SPLINE
SPL {X  -140.007, Y  +297.383, Z    +0.000, E1   +42.766, E3 +239231.187}
SPL {X  -156.919, Y  +337.064, Z    +0.000, E1   +27.647, E3 +239237.338}
SPL {X  -160.736, Y  +354.534, Z    +0.000, E1   +18.553, E3 +239240.033}
SPL {X  -162.078, Y  +364.978, Z    +0.000, E1   +12.369, E3 +239241.718}
SPL {X  -162.752, Y  +375.778, Z    +0.000, E1    +5.236, E3 +239241.427}
SPL {X  -162.820, Y  +381.939, Z    +0.000, E1    +0.593, E3 +239241.054}
SPL {X  -162.820, Y  +383.993, Z    +0.000, E1    -1.497, E3 +239240.627}
SPL {X  -162.820, Y  +388.628, Z    +0.000, E1    -7.678, E3 +239240.530}
SPL {X  -162.820, Y  +394.643, Z    +0.000, E1   -17.317, E3 +239240.330}
SPL {X  -162.820, Y  +401.515, Z    +0.000, E1   -27.960, E3 +239241.150}
SPL {X  -162.820, Y  +415.147, Z    +0.000, E1   -45.856, E3 +239240.466}
SPL {X  -162.820, Y  +437.881, Z    +0.000, E1   -59.335, E3 +239245.884}
SPL {X  -162.820, Y  +475.967, Z    +0.000, E1   -65.140, E3 +239263.337}
SPL {X  -162.820, Y  +578.686, Z    +0.000, E1   -67.085, E3 +239331.578}
ENDSPLINE

SPLINE
SPL {X  -162.820, Y  +565.364, Z    +0.000, E1   -63.589, E3 +239345.578}
ENDSPLINE

SPLINE
SPL {X  -162.820, Y  +574.608, Z    +0.000, E1   -63.370, E3 +239356.837}
SPL {X  -162.820, Y  +584.314, Z    +0.000, E1   -63.342, E3 +239367.129}
SPL {X  -162.820, Y  +593.857, Z    +0.000, E1   -63.382, E3 +239376.831}
SPL {X  -162.820, Y  +602.272, Z    +0.000, E1   -63.279, E3 +239386.359}
SPL {X  -162.820, Y  +613.309, Z    +0.000, E1   -63.489, E3 +239396.358}
SPL {X  -162.820, Y  +619.956, Z    +0.000, E1   -63.110, E3 +239406.044}
SPL {X  -162.820, Y  +634.513, Z    +0.000, E1   -63.471, E3 +239418.810}
SPL {X  -162.820, Y  +648.936, Z    +0.000, E1   -63.278, E3 +239435.265}
SPL {X  -162.820, Y  +662.662, Z    +0.000, E1   -63.383, E3 +239448.757}
SPL {X  -162.819, Y  +673.983, Z    +0.000, E1   -63.398, E3 +239460.480}
SPL {X  -162.399, Y  +685.202, Z    +0.000, E1   -63.235, E3 +239473.474}
SPL {X  -161.289, Y  +695.772, Z    +0.000, E1   -63.167, E3 +239484.924}
SPL {X  -160.212, Y  +702.527, Z    +0.000, E1   -62.898, E3 +239493.905}
SPL {X  -158.647, Y  +710.128, Z    +0.000, E1   -62.776, E3 +239502.727}
SPL {X  -156.957, Y  +716.799, Z    +0.000, E1   -62.460, E3 +239511.845}
SPL {X  -154.447, Y  +725.041, Z    +0.000, E1   -62.170, E3 +239522.503}
SPL {X  -151.721, Y  +732.586, Z    +0.000, E1   -61.616, E3 +239533.752}
SPL {X  -149.420, Y  +738.185, Z    +0.000, E1   -61.282, E3 +239541.642}
SPL {X  -146.033, Y  +745.504, Z    +0.000, E1   -60.844, E3 +239551.909}
SPL {X  -142.518, Y  +752.234, Z    +0.000, E1   -60.144, E3 +239562.535}
SPL {X  -139.430, Y  +757.582, Z    +0.000, E1   -59.554, E3 +239571.067}
SPL {X  -134.550, Y  +765.187, Z    +0.000, E1   -59.954, E3 +239577.018}
SPL {X  -102.851, Y  +799.722, Z    +0.000, E1   -53.923, E3 +239667.511}
SPL {X  -101.618, Y  +800.716, Z    +0.000, E1   -52.212, E3 +239780.496}
ENDSPLINE

SPLINE
SPL {X  -141.567, Y  +753.931, Z    +0.000, E1   -42.659, E3 +239817.198}
SPL {X  -155.442, Y  +721.958, Z    +0.000, E1   -30.769, E3 +239824.104}
SPL {X  -161.417, Y  +694.832, Z    +0.000, E1   -16.464, E3 +239828.073}
SPL {X  -162.580, Y  +682.344, Z    +0.000, E1    -8.212, E3 +239828.280}
SPL {X  -162.811, Y  +675.182, Z    +0.000, E1    -3.078, E3 +239828.313}
SPL {X  -162.820, Y  +671.474, Z    +0.000, E1    -0.022, E3 +239827.783}
SPL {X  -162.820, Y  +668.525, Z    +0.000, E1    +3.543, E3 +239827.476}
SPL {X  -162.820, Y  +663.189, Z    +0.000, E1   +11.952, E3 +239827.465}
SPL {X  -162.820, Y  +655.445, Z    +0.000, E1   +24.952, E3 +239827.412}
SPL {X  -162.820, Y  +644.088, Z    +0.000, E1   +41.840, E3 +239827.548}
SPL {X  -162.820, Y  +632.645, Z    +0.000, E1   +53.114, E3 +239828.283}
SPL {X  -162.820, Y  +584.142, Z    +0.000, E1   +66.966, E3 +239843.626}
SPL {X  -162.820, Y  +471.906, Z    +0.000, E1   +66.781, E3 +239925.868}
SPL {X  -162.820, Y  +470.218, Z    +0.000, E1   +64.979, E3 +239941.868}
SPL {X  -162.820, Y  +452.619, Z    +0.000, E1   +64.912, E3 +239959.546}
SPL {X  -162.820, Y  +437.579, Z    +0.000, E1   +64.893, E3 +239974.228}
SPL {X  -162.820, Y  +425.248, Z    +0.000, E1   +64.950, E3 +239985.816}
SPL {X  -162.820, Y  +417.868, Z    +0.000, E1   +64.478, E3 +239996.634}
ENDSPLINE

SPLINE
SPL {X  -162.820, Y  +442.889, Z    +0.000, E1   +58.918, E3 +240008.814}
ENDSPLINE

SPLINE
SPL {X  -162.820, Y  +428.091, Z    +0.000, E1   +59.583, E3 +240022.587}
SPL {X  -162.820, Y  +410.436, Z    +0.000, E1   +60.611, E3 +240036.788}
SPL {X  -162.820, Y  +385.611, Z    +0.000, E1   +62.089, E3 +240054.686}
ENDSPLINE

SPLINE
SPL {X  -162.820, Y  +397.122, Z    +0.000, E1   +58.099, E3 +240067.658}
ENDSPLINE

SPLINE
SPL {X  -162.820, Y  +387.359, Z    +0.000, E1   +58.365, E3 +240078.519}
SPL {X  -162.810, Y  +378.731, Z    +0.000, E1   +58.366, E3 +240089.577}
SPL {X  -162.546, Y  +371.051, Z    +0.000, E1   +58.239, E3 +240100.297}
SPL {X  -161.863, Y  +362.875, Z    +0.000, E1   +58.273, E3 +240110.522}
SPL {X  -161.159, Y  +357.301, Z    +0.000, E1   +57.946, E3 +240119.822}
SPL {X  -159.864, Y  +349.614, Z    +0.000, E1   +57.922, E3 +240129.898}
SPL {X  -158.300, Y  +342.404, Z    +0.000, E1   +57.579, E3 +240141.344}
SPL {X  -156.187, Y  +334.499, Z    +0.000, E1   +57.331, E3 +240153.004}
SPL {X  -154.237, Y  +328.333, Z    +0.000, E1   +56.930, E3 +240163.214}
SPL {X  -152.732, Y  +324.078, Z    +0.000, E1   +56.482, E3 +240171.219}
SPL {X  -150.609, Y  +318.634, Z    +0.000, E1   +56.366, E3 +240178.913}
SPL {X  -148.206, Y  +313.080, Z    +0.000, E1   +55.888, E3 +240188.625}
SPL {X  -145.956, Y  +308.339, Z    +0.000, E1   +55.380, E3 +240197.301}
SPL {X  -143.330, Y  +303.254, Z    +0.000, E1   +55.057, E3 +240205.421}
SPL {X  -137.431, Y  +293.190, Z    +0.000, E1   +56.809, E3 +240209.584}
SPL {X  -115.845, Y  +266.087, Z    +0.000, E1   +50.276, E3 +240308.442}
SPL {X  -114.083, Y  +264.330, Z    +0.000, E1   +49.123, E3 +240347.152}
ENDSPLINE

SPLINE
SPL {X  -149.622, Y  +316.285, Z    +0.000, E1   +35.036, E3 +240415.664}
SPL {X  -158.704, Y  +344.121, Z    +0.000, E1   +23.312, E3 +240425.537}
SPL {X  -161.701, Y  +361.440, Z    +0.000, E1   +13.961, E3 +240424.608}
SPL {X  -162.691, Y  +374.019, Z    +0.000, E1    +6.263, E3 +240425.261}
SPL {X  -162.820, Y  +381.771, Z    +0.000, E1    +0.850, E3 +240424.745}
SPL {X  -162.820, Y  +384.317, Z    +0.000, E1    -1.618, E3 +240424.463}
SPL {X  -162.820, Y  +387.033, Z    +0.000, E1    -4.758, E3 +240424.255}
SPL {X  -162.820, Y  +390.967, Z    +0.000, E1    -9.918, E3 +240424.700}
SPL {X  -162.820, Y  +395.392, Z    +0.000, E1   -16.726, E3 +240423.141}
SPL {X  -162.820, Y  +402.654, Z    +0.000, E1   -26.492, E3 +240425.032}
SPL {X  -162.820, Y  +417.515, Z    +0.000, E1   -44.878, E3 +240424.149}
SPL {X  -162.820, Y  +462.065, Z    +0.000, E1   -61.507, E3 +240441.109}
SPL {X  -162.820, Y  +504.602, Z    +0.000, E1   -64.286, E3 +240466.635}
SPL {X  -162.820, Y  +535.709, Z    +0.000, E1   -59.182, E3 +240524.314}
SPL {X  -162.820, Y  +543.678, Z    +0.000, E1   -58.515, E3 +240538.703}
SPL {X  -162.820, Y  +553.725, Z    +0.000, E1   -58.454, E3 +240551.964}
SPL {X  -162.820, Y  +562.850, Z    +0.000, E1   -58.373, E3 +240564.126}
SPL {X  -162.820, Y  +573.452, Z    +0.000, E1   -58.444, E3 +240577.339}
SPL {X  -162.820, Y  +583.632, Z    +0.000, E1   -58.444, E3 +240590.266}
SPL {X  -162.820, Y  +591.768, Z    +0.000, E1   -58.375, E3 +240601.130}
SPL {X  -162.820, Y  +601.090, Z    +0.000, E1   -58.519, E3 +240612.117}
SPL {X  -162.820, Y  +609.492, Z    +0.000, E1   -58.431, E3 +240623.422}
SPL {X  -162.820, Y  +617.241, Z    +0.000, E1   -58.340, E3 +240633.947}
SPL {X  -162.820, Y  +626.506, Z    +0.000, E1   -58.420, E3 +240645.329}
SPL {X  -162.820, Y  +635.919, Z    +0.000, E1   -58.604, E3 +240656.073}
SPL {X  -162.820, Y  +643.895, Z    +0.000, E1   -58.380, E3 +240667.838}
SPL {X  -162.820, Y  +653.118, Z    +0.000, E1   -58.401, E3 +240679.435}
SPL {X  -162.820, Y  +660.924, Z    +0.000, E1   -58.393, E3 +240689.503}
SPL {X  -162.820, Y  +670.459, Z    +0.000, E1   -58.489, E3 +240701.104}
SPL {X  -162.713, Y  +679.396, Z    +0.000, E1   -58.414, E3 +240713.003}
SPL {X  -162.301, Y  +686.495, Z    +0.000, E1   -58.302, E3 +240722.787}
SPL {X  -161.571, Y  +693.631, Z    +0.000, E1   -58.186, E3 +240732.751}
SPL {X  -160.411, Y  +701.402, Z    +0.000, E1   -58.100, E3 +240743.227}
SPL {X  -159.229, Y  +707.508, Z    +0.000, E1   -57.870, E3 +240752.465}
SPL {X  -157.825, Y  +713.519, Z    +0.000, E1   -57.630, E3 +240761.701}
SPL {X  -156.079, Y  +719.864, Z    +0.000, E1   -57.324, E3 +240771.664}
SPL {X  -154.064, Y  +726.175, Z    +0.000, E1   -57.042, E3 +240781.426}
SPL {X  -152.053, Y  +731.726, Z    +0.000, E1   -56.648, E3 +240790.711}
SPL {X  -150.108, Y  +736.570, Z    +0.000, E1   -56.283, E3 +240798.950}
SPL {X  -147.726, Y  +741.964, Z    +0.000, E1   -55.884, E3 +240807.986}
SPL {X  -145.163, Y  +747.242, Z    +0.000, E1   -55.517, E3 +240816.582}
SPL {X  -142.489, Y  +752.286, Z    +0.000, E1   -55.227, E3 +240824.409}
SPL {X  -136.074, Y  +762.910, Z    +0.000, E1   -57.336, E3 +240827.531}
SPL {X  -116.561, Y  +787.183, Z    +0.000, E1   -51.088, E3 +240911.999}
ENDSPLINE

SPLINE
SPL {X  -119.623, Y  +783.957, Z    +0.000, E1   -49.202, E3 +241036.532}
SPL {X  -149.958, Y  +736.927, Z    +0.000, E1   -34.772, E3 +241034.249}
SPL {X  -158.826, Y  +709.343, Z    +0.000, E1   -23.029, E3 +241042.592}
SPL {X  -161.344, Y  +695.370, Z    +0.000, E1   -15.607, E3 +241044.991}
SPL {X  -162.477, Y  +684.065, Z    +0.000, E1    -8.887, E3 +241044.621}
SPL {X  -162.813, Y  +675.055, Z    +0.000, E1    -2.911, E3 +241045.184}
SPL {X  -162.820, Y  +670.901, Z    +0.000, E1    +0.338, E3 +241044.555}
SPL {X  -162.820, Y  +667.984, Z    +0.000, E1    +3.594, E3 +241044.387}
SPL {X  -162.820, Y  +664.667, Z    +0.000, E1    +7.867, E3 +241044.100}
SPL {X  -162.820, Y  +660.022, Z    +0.000, E1   +14.535, E3 +241043.997}
SPL {X  -162.820, Y  +653.408, Z    +0.000, E1   +24.221, E3 +241044.307}
SPL {X  -162.820, Y  +640.244, Z    +0.000, E1   +41.042, E3 +241044.351}
SPL {X  -162.820, Y  +592.517, Z    +0.000, E1   +60.575, E3 +241063.482}
SPL {X  -162.820, Y  +515.613, Z    +0.000, E1   +60.751, E3 +241137.317}
ENDSPLINE

SPLINE
SPL {X  -162.820, Y  +518.198, Z    +0.000, E1   +58.338, E3 +241150.473}
ENDSPLINE

SPLINE
SPL {X  -162.820, Y  +508.314, Z    +0.000, E1   +58.337, E3 +241163.169}
SPL {X  -162.820, Y  +498.518, Z    +0.000, E1   +58.346, E3 +241175.675}
SPL {X  -162.820, Y  +489.418, Z    +0.000, E1   +58.357, E3 +241187.265}
SPL {X  -162.820, Y  +479.904, Z    +0.000, E1   +58.389, E3 +241199.312}
SPL {X  -162.820, Y  +472.095, Z    +0.000, E1   +58.202, E3 +241210.492}
SPL {X  -162.820, Y  +463.661, Z    +0.000, E1   +58.370, E3 +241220.278}
SPL {X  -162.820, Y  +454.904, Z    +0.000, E1   +58.380, E3 +241231.444}
SPL {X  -162.820, Y  +446.206, Z    +0.000, E1   +58.278, E3 +241243.335}
SPL {X  -162.820, Y  +436.416, Z    +0.000, E1   +58.325, E3 +241255.575}
SPL {X  -162.820, Y  +426.628, Z    +0.000, E1   +58.432, E3 +241267.443}
SPL {X  -162.820, Y  +418.389, Z    +0.000, E1   +58.300, E3 +241278.846}
SPL {X  -162.820, Y  +412.292, Z    +0.000, E1   +58.070, E3 +241288.214}
SPL {X  -162.820, Y  +403.663, Z    +0.000, E1   +58.258, E3 +241298.154}
SPL {X  -162.820, Y  +397.157, Z    +0.000, E1   +58.054, E3 +241307.890}
SPL {X  -162.820, Y  +387.359, Z    +0.000, E1   +58.365, E3 +241318.519}
SPL {X  -162.810, Y  +378.731, Z    +0.000, E1   +58.366, E3 +241329.577}
SPL {X  -162.546, Y  +371.051, Z    +0.000, E1   +58.239, E3 +241340.297}
SPL {X  -161.863, Y  +362.875, Z    +0.000, E1   +58.273, E3 +241350.522}
SPL {X  -161.159, Y  +357.301, Z    +0.000, E1   +57.946, E3 +241359.822}
SPL {X  -159.864, Y  +349.614, Z    +0.000, E1   +57.922, E3 +241369.898}
SPL {X  -158.300, Y  +342.404, Z    +0.000, E1   +57.579, E3 +241381.344}
SPL {X  -156.187, Y  +334.499, Z    +0.000, E1   +57.331, E3 +241393.004}
SPL {X  -154.237, Y  +328.333, Z    +0.000, E1   +56.930, E3 +241403.214}
SPL {X  -152.732, Y  +324.078, Z    +0.000, E1   +56.482, E3 +241411.219}
SPL {X  -150.609, Y  +318.634, Z    +0.000, E1   +56.366, E3 +241418.913}
SPL {X  -148.206, Y  +313.080, Z    +0.000, E1   +55.888, E3 +241428.625}
SPL {X  -145.956, Y  +308.339, Z    +0.000, E1   +55.380, E3 +241437.301}
SPL {X  -143.330, Y  +303.254, Z    +0.000, E1   +55.057, E3 +241445.421}
SPL {X  -137.431, Y  +293.190, Z    +0.000, E1   +56.809, E3 +241449.584}
SPL {X  -115.845, Y  +266.087, Z    +0.000, E1   +50.276, E3 +241548.442}
SPL {X  -114.083, Y  +264.330, Z    +0.000, E1   +49.123, E3 +241587.152}
ENDSPLINE

SPLINE
SPL {X  -149.622, Y  +316.285, Z    +0.000, E1   +35.036, E3 +241655.664}
SPL {X  -158.704, Y  +344.121, Z    +0.000, E1   +23.312, E3 +241665.537}
SPL {X  -161.701, Y  +361.440, Z    +0.000, E1   +13.961, E3 +241664.608}
SPL {X  -162.691, Y  +374.019, Z    +0.000, E1    +6.263, E3 +241665.261}
SPL {X  -162.820, Y  +380.238, Z    +0.000, E1    +1.925, E3 +241664.945}
SPL {X  -162.820, Y  +382.545, Z    +0.000, E1    +0.100, E3 +241664.644}
SPL {X  -162.820, Y  +384.317, Z    +0.000, E1    -1.618, E3 +241664.463}
SPL {X  -162.820, Y  +387.033, Z    +0.000, E1    -4.758, E3 +241664.255}
SPL {X  -162.820, Y  +390.967, Z    +0.000, E1    -9.918, E3 +241664.700}
SPL {X  -162.820, Y  +395.392, Z    +0.000, E1   -16.726, E3 +241663.141}
SPL {X  -162.820, Y  +402.654, Z    +0.000, E1   -26.492, E3 +241665.032}
SPL {X  -162.820, Y  +417.515, Z    +0.000, E1   -44.878, E3 +241664.149}
SPL {X  -162.820, Y  +462.065, Z    +0.000, E1   -61.507, E3 +241681.109}
SPL {X  -162.820, Y  +504.602, Z    +0.000, E1   -64.286, E3 +241706.635}
SPL {X  -162.820, Y  +539.530, Z    +0.000, E1   -60.821, E3 +241757.326}
ENDSPLINE

SPLINE
SPL {X  -162.820, Y  +534.172, Z    +0.000, E1   -58.470, E3 +241766.826}
ENDSPLINE

SPLINE
SPL {X  -162.820, Y  +543.678, Z    +0.000, E1   -58.515, E3 +241778.703}
SPL {X  -162.820, Y  +553.725, Z    +0.000, E1   -58.454, E3 +241791.964}
SPL {X  -162.820, Y  +562.850, Z    +0.000, E1   -58.373, E3 +241804.126}
SPL {X  -162.820, Y  +571.217, Z    +0.000, E1   -58.397, E3 +241814.679}
SPL {X  -162.820, Y  +581.879, Z    +0.000, E1   -58.475, E3 +241827.932}
SPL {X  -162.820, Y  +591.768, Z    +0.000, E1   -58.375, E3 +241841.130}
SPL {X  -162.820, Y  +601.090, Z    +0.000, E1   -58.519, E3 +241852.117}
SPL {X  -162.820, Y  +609.492, Z    +0.000, E1   -58.431, E3 +241863.422}
SPL {X  -162.820, Y  +617.241, Z    +0.000, E1   -58.340, E3 +241873.947}
SPL {X  -162.820, Y  +626.506, Z    +0.000, E1   -58.420, E3 +241885.329}
SPL {X  -162.820, Y  +635.919, Z    +0.000, E1   -58.604, E3 +241896.073}
SPL {X  -162.820, Y  +643.895, Z    +0.000, E1   -58.380, E3 +241907.838}
SPL {X  -162.820, Y  +653.118, Z    +0.000, E1   -58.401, E3 +241919.435}
SPL {X  -162.820, Y  +660.924, Z    +0.000, E1   -58.393, E3 +241929.503}
SPL {X  -162.820, Y  +670.459, Z    +0.000, E1   -58.489, E3 +241941.104}
SPL {X  -162.713, Y  +679.396, Z    +0.000, E1   -58.414, E3 +241953.003}
SPL {X  -162.301, Y  +686.495, Z    +0.000, E1   -58.302, E3 +241962.787}
SPL {X  -161.571, Y  +693.631, Z    +0.000, E1   -58.186, E3 +241972.751}
SPL {X  -160.411, Y  +701.402, Z    +0.000, E1   -58.100, E3 +241983.227}
SPL {X  -159.229, Y  +707.508, Z    +0.000, E1   -57.870, E3 +241992.465}
SPL {X  -157.825, Y  +713.519, Z    +0.000, E1   -57.630, E3 +242001.701}
SPL {X  -156.079, Y  +719.864, Z    +0.000, E1   -57.324, E3 +242011.664}
SPL {X  -154.064, Y  +726.175, Z    +0.000, E1   -57.042, E3 +242021.426}
SPL {X  -152.053, Y  +731.726, Z    +0.000, E1   -56.648, E3 +242030.711}
SPL {X  -150.108, Y  +736.570, Z    +0.000, E1   -56.283, E3 +242038.950}
SPL {X  -147.726, Y  +741.964, Z    +0.000, E1   -55.884, E3 +242047.986}
SPL {X  -145.163, Y  +747.242, Z    +0.000, E1   -55.517, E3 +242056.582}
SPL {X  -142.489, Y  +752.286, Z    +0.000, E1   -55.227, E3 +242064.409}
SPL {X  -136.074, Y  +762.910, Z    +0.000, E1   -57.336, E3 +242067.531}
SPL {X  -116.561, Y  +787.183, Z    +0.000, E1   -51.088, E3 +242151.999}
ENDSPLINE

SPLINE
SPL {X  -119.623, Y  +783.957, Z    +0.000, E1   -49.202, E3 +242276.532}
SPL {X  -149.958, Y  +736.927, Z    +0.000, E1   -34.772, E3 +242274.249}
SPL {X  -158.826, Y  +709.343, Z    +0.000, E1   -23.029, E3 +242282.592}
SPL {X  -161.800, Y  +691.694, Z    +0.000, E1   -13.520, E3 +242284.886}
SPL {X  -162.711, Y  +679.444, Z    +0.000, E1    -5.922, E3 +242284.960}
SPL {X  -162.820, Y  +672.303, Z    +0.000, E1    -0.875, E3 +242284.825}
SPL {X  -162.820, Y  +669.030, Z    +0.000, E1    +2.242, E3 +242284.397}
SPL {X  -162.820, Y  +664.667, Z    +0.000, E1    +7.867, E3 +242284.100}
SPL {X  -162.820, Y  +660.022, Z    +0.000, E1   +14.535, E3 +242283.997}
SPL {X  -162.820, Y  +653.408, Z    +0.000, E1   +24.221, E3 +242284.307}
SPL {X  -162.820, Y  +640.244, Z    +0.000, E1   +41.042, E3 +242284.351}
SPL {X  -162.820, Y  +592.517, Z    +0.000, E1   +60.575, E3 +242303.482}
SPL {X  -162.820, Y  +515.613, Z    +0.000, E1   +60.751, E3 +242377.317}
ENDSPLINE

SPLINE
SPL {X  -162.820, Y  +518.198, Z    +0.000, E1   +58.338, E3 +242390.473}
ENDSPLINE

SPLINE
SPL {X  -162.820, Y  +508.314, Z    +0.000, E1   +58.337, E3 +242403.169}
SPL {X  -162.820, Y  +498.518, Z    +0.000, E1   +58.346, E3 +242415.675}
SPL {X  -162.820, Y  +489.418, Z    +0.000, E1   +58.357, E3 +242427.265}
SPL {X  -162.820, Y  +479.904, Z    +0.000, E1   +58.389, E3 +242439.312}
SPL {X  -162.820, Y  +472.095, Z    +0.000, E1   +58.202, E3 +242450.492}
SPL {X  -162.820, Y  +463.661, Z    +0.000, E1   +58.370, E3 +242460.278}
SPL {X  -162.820, Y  +454.904, Z    +0.000, E1   +58.380, E3 +242471.444}
SPL {X  -162.820, Y  +446.206, Z    +0.000, E1   +58.278, E3 +242483.335}
SPL {X  -162.820, Y  +436.416, Z    +0.000, E1   +58.325, E3 +242495.575}
SPL {X  -162.820, Y  +426.628, Z    +0.000, E1   +58.432, E3 +242507.443}
SPL {X  -162.820, Y  +418.389, Z    +0.000, E1   +58.300, E3 +242518.846}
SPL {X  -162.820, Y  +412.292, Z    +0.000, E1   +58.070, E3 +242528.214}
SPL {X  -162.820, Y  +403.663, Z    +0.000, E1   +58.258, E3 +242538.154}
SPL {X  -162.820, Y  +397.157, Z    +0.000, E1   +58.054, E3 +242547.890}
SPL {X  -162.820, Y  +387.359, Z    +0.000, E1   +58.365, E3 +242558.519}
SPL {X  -162.810, Y  +378.731, Z    +0.000, E1   +58.366, E3 +242569.577}
SPL {X  -162.546, Y  +371.051, Z    +0.000, E1   +58.239, E3 +242580.297}
SPL {X  -161.863, Y  +362.875, Z    +0.000, E1   +58.273, E3 +242590.522}
SPL {X  -161.159, Y  +357.301, Z    +0.000, E1   +57.946, E3 +242599.822}
SPL {X  -159.864, Y  +349.614, Z    +0.000, E1   +57.922, E3 +242609.898}
SPL {X  -158.548, Y  +343.449, Z    +0.000, E1   +57.711, E3 +242619.072}
SPL {X  -156.580, Y  +335.856, Z    +0.000, E1   +57.340, E3 +242631.295}
SPL {X  -154.237, Y  +328.333, Z    +0.000, E1   +56.930, E3 +242643.214}
SPL {X  -152.732, Y  +324.078, Z    +0.000, E1   +56.482, E3 +242651.219}
SPL {X  -150.609, Y  +318.634, Z    +0.000, E1   +56.366, E3 +242658.913}
SPL {X  -148.206, Y  +313.080, Z    +0.000, E1   +55.888, E3 +242668.625}
SPL {X  -145.956, Y  +308.339, Z    +0.000, E1   +55.380, E3 +242677.301}
SPL {X  -143.330, Y  +303.254, Z    +0.000, E1   +55.057, E3 +242685.421}
SPL {X  -137.431, Y  +293.190, Z    +0.000, E1   +56.809, E3 +242689.584}
SPL {X  -115.845, Y  +266.087, Z    +0.000, E1   +50.276, E3 +242788.442}
SPL {X  -114.083, Y  +264.330, Z    +0.000, E1   +49.123, E3 +242827.152}
ENDSPLINE

SPLINE
SPL {X  -149.622, Y  +316.285, Z    +0.000, E1   +35.036, E3 +242895.664}
SPL {X  -158.704, Y  +344.121, Z    +0.000, E1   +23.312, E3 +242905.537}
SPL {X  -161.701, Y  +361.440, Z    +0.000, E1   +13.961, E3 +242904.608}
SPL {X  -162.691, Y  +374.019, Z    +0.000, E1    +6.263, E3 +242905.261}
SPL {X  -162.820, Y  +381.771, Z    +0.000, E1    +0.850, E3 +242904.745}
SPL {X  -162.820, Y  +384.317, Z    +0.000, E1    -1.618, E3 +242904.463}
SPL {X  -162.820, Y  +387.033, Z    +0.000, E1    -4.758, E3 +242904.255}
SPL {X  -162.820, Y  +390.967, Z    +0.000, E1    -9.918, E3 +242904.700}
SPL {X  -162.820, Y  +395.392, Z    +0.000, E1   -16.726, E3 +242903.141}
SPL {X  -162.820, Y  +402.654, Z    +0.000, E1   -26.492, E3 +242905.032}
SPL {X  -162.820, Y  +417.515, Z    +0.000, E1   -44.878, E3 +242904.149}
SPL {X  -162.820, Y  +462.065, Z    +0.000, E1   -61.507, E3 +242921.109}
SPL {X  -162.820, Y  +504.602, Z    +0.000, E1   -64.286, E3 +242946.635}
SPL {X  -162.820, Y  +539.530, Z    +0.000, E1   -60.821, E3 +242997.326}
ENDSPLINE

SPLINE
SPL {X  -162.820, Y  +534.172, Z    +0.000, E1   -58.470, E3 +243006.826}
ENDSPLINE

SPLINE
SPL {X  -162.820, Y  +543.678, Z    +0.000, E1   -58.515, E3 +243018.703}
SPL {X  -162.820, Y  +553.725, Z    +0.000, E1   -58.454, E3 +243031.964}
SPL {X  -162.820, Y  +562.850, Z    +0.000, E1   -58.373, E3 +243044.126}
SPL {X  -162.820, Y  +571.217, Z    +0.000, E1   -58.397, E3 +243054.679}
SPL {X  -162.820, Y  +581.879, Z    +0.000, E1   -58.475, E3 +243067.932}
SPL {X  -162.820, Y  +591.768, Z    +0.000, E1   -58.375, E3 +243081.130}
SPL {X  -162.820, Y  +601.090, Z    +0.000, E1   -58.519, E3 +243092.117}
SPL {X  -162.820, Y  +609.492, Z    +0.000, E1   -58.431, E3 +243103.422}
SPL {X  -162.820, Y  +617.241, Z    +0.000, E1   -58.340, E3 +243113.947}
SPL {X  -162.820, Y  +626.506, Z    +0.000, E1   -58.420, E3 +243125.329}
SPL {X  -162.820, Y  +638.850, Z    +0.000, E1   -58.527, E3 +243140.545}
SPL {X  -162.820, Y  +651.112, Z    +0.000, E1   -58.411, E3 +243156.903}
SPL {X  -162.820, Y  +660.924, Z    +0.000, E1   -58.393, E3 +243169.503}
SPL {X  -162.820, Y  +670.459, Z    +0.000, E1   -58.489, E3 +243181.104}
SPL {X  -162.713, Y  +679.396, Z    +0.000, E1   -58.414, E3 +243193.003}
SPL {X  -162.301, Y  +686.495, Z    +0.000, E1   -58.302, E3 +243202.787}
SPL {X  -161.571, Y  +693.631, Z    +0.000, E1   -58.186, E3 +243212.751}
SPL {X  -160.411, Y  +701.402, Z    +0.000, E1   -58.100, E3 +243223.227}
SPL {X  -159.229, Y  +707.508, Z    +0.000, E1   -57.870, E3 +243232.465}
SPL {X  -157.825, Y  +713.519, Z    +0.000, E1   -57.630, E3 +243241.701}
SPL {X  -156.079, Y  +719.864, Z    +0.000, E1   -57.324, E3 +243251.664}
SPL {X  -154.064, Y  +726.175, Z    +0.000, E1   -57.042, E3 +243261.426}
SPL {X  -152.053, Y  +731.726, Z    +0.000, E1   -56.648, E3 +243270.711}
SPL {X  -150.108, Y  +736.570, Z    +0.000, E1   -56.283, E3 +243278.950}
SPL {X  -147.726, Y  +741.964, Z    +0.000, E1   -55.884, E3 +243287.986}
SPL {X  -145.163, Y  +747.242, Z    +0.000, E1   -55.517, E3 +243296.582}
SPL {X  -142.489, Y  +752.286, Z    +0.000, E1   -55.227, E3 +243304.409}
SPL {X  -136.074, Y  +762.910, Z    +0.000, E1   -57.336, E3 +243307.531}
SPL {X  -116.561, Y  +787.183, Z    +0.000, E1   -51.088, E3 +243391.999}
ENDSPLINE

SPLINE
SPL {X  -119.623, Y  +783.957, Z    +0.000, E1   -49.202, E3 +243516.532}
SPL {X  -149.958, Y  +736.927, Z    +0.000, E1   -34.772, E3 +243514.249}
SPL {X  -158.826, Y  +709.343, Z    +0.000, E1   -23.029, E3 +243522.592}
SPL {X  -161.344, Y  +695.370, Z    +0.000, E1   -15.607, E3 +243524.991}
SPL {X  -162.477, Y  +684.065, Z    +0.000, E1    -8.887, E3 +243524.621}
SPL {X  -162.813, Y  +675.055, Z    +0.000, E1    -2.911, E3 +243525.184}
SPL {X  -162.820, Y  +670.901, Z    +0.000, E1    +0.338, E3 +243524.555}
SPL {X  -162.820, Y  +667.984, Z    +0.000, E1    +3.594, E3 +243524.387}
SPL {X  -162.820, Y  +664.667, Z    +0.000, E1    +7.867, E3 +243524.100}
SPL {X  -162.820, Y  +660.022, Z    +0.000, E1   +14.535, E3 +243523.997}
SPL {X  -162.820, Y  +653.408, Z    +0.000, E1   +24.221, E3 +243524.307}
SPL {X  -162.820, Y  +640.244, Z    +0.000, E1   +41.042, E3 +243524.351}
SPL {X  -162.820, Y  +592.517, Z    +0.000, E1   +60.575, E3 +243543.482}
SPL {X  -162.820, Y  +515.613, Z    +0.000, E1   +60.751, E3 +243617.317}
ENDSPLINE

SPLINE
SPL {X  -162.820, Y  +518.198, Z    +0.000, E1   +58.338, E3 +243630.473}
ENDSPLINE

SPLINE
SPL {X  -162.820, Y  +508.314, Z    +0.000, E1   +58.337, E3 +243643.169}
SPL {X  -162.820, Y  +498.518, Z    +0.000, E1   +58.346, E3 +243655.675}
SPL {X  -162.820, Y  +489.418, Z    +0.000, E1   +58.357, E3 +243667.265}
SPL {X  -162.820, Y  +479.904, Z    +0.000, E1   +58.389, E3 +243679.312}
SPL {X  -162.820, Y  +472.095, Z    +0.000, E1   +58.202, E3 +243690.492}
SPL {X  -162.820, Y  +463.661, Z    +0.000, E1   +58.370, E3 +243700.278}
SPL {X  -162.820, Y  +454.904, Z    +0.000, E1   +58.380, E3 +243711.444}
SPL {X  -162.820, Y  +446.206, Z    +0.000, E1   +58.278, E3 +243723.335}
SPL {X  -162.820, Y  +436.416, Z    +0.000, E1   +58.325, E3 +243735.575}
SPL {X  -162.820, Y  +426.628, Z    +0.000, E1   +58.432, E3 +243747.443}
SPL {X  -162.820, Y  +418.389, Z    +0.000, E1   +58.300, E3 +243758.846}
SPL {X  -162.820, Y  +412.292, Z    +0.000, E1   +58.070, E3 +243768.214}
SPL {X  -162.820, Y  +403.663, Z    +0.000, E1   +58.258, E3 +243778.154}
SPL {X  -162.820, Y  +397.157, Z    +0.000, E1   +58.054, E3 +243787.890}
SPL {X  -162.820, Y  +387.359, Z    +0.000, E1   +58.365, E3 +243798.519}
SPL {X  -162.810, Y  +378.731, Z    +0.000, E1   +58.366, E3 +243809.577}
SPL {X  -162.546, Y  +371.051, Z    +0.000, E1   +58.239, E3 +243820.297}
SPL {X  -161.863, Y  +362.875, Z    +0.000, E1   +58.273, E3 +243830.522}
SPL {X  -161.159, Y  +357.301, Z    +0.000, E1   +57.946, E3 +243839.822}
SPL {X  -159.864, Y  +349.614, Z    +0.000, E1   +57.922, E3 +243849.898}
SPL {X  -158.300, Y  +342.404, Z    +0.000, E1   +57.579, E3 +243861.344}
SPL {X  -156.187, Y  +334.499, Z    +0.000, E1   +57.331, E3 +243873.004}
SPL {X  -154.237, Y  +328.333, Z    +0.000, E1   +56.930, E3 +243883.214}
SPL {X  -152.732, Y  +324.078, Z    +0.000, E1   +56.482, E3 +243891.219}
SPL {X  -150.609, Y  +318.634, Z    +0.000, E1   +56.366, E3 +243898.913}
SPL {X  -148.206, Y  +313.080, Z    +0.000, E1   +55.888, E3 +243908.625}
SPL {X  -145.956, Y  +308.339, Z    +0.000, E1   +55.380, E3 +243917.301}
SPL {X  -143.330, Y  +303.254, Z    +0.000, E1   +55.057, E3 +243925.421}
SPL {X  -137.431, Y  +293.190, Z    +0.000, E1   +56.809, E3 +243929.584}
SPL {X  -115.845, Y  +266.087, Z    +0.000, E1   +50.276, E3 +244028.442}
SPL {X  -114.083, Y  +264.330, Z    +0.000, E1   +49.123, E3 +244067.152}
ENDSPLINE

SPLINE
SPL {X  -149.622, Y  +316.285, Z    +0.000, E1   +35.036, E3 +244135.664}
SPL {X  -158.704, Y  +344.121, Z    +0.000, E1   +23.312, E3 +244145.537}
SPL {X  -161.701, Y  +361.440, Z    +0.000, E1   +13.961, E3 +244144.608}
SPL {X  -162.691, Y  +374.019, Z    +0.000, E1    +6.263, E3 +244145.261}
SPL {X  -162.820, Y  +381.771, Z    +0.000, E1    +0.850, E3 +244144.745}
SPL {X  -162.820, Y  +384.317, Z    +0.000, E1    -1.618, E3 +244144.463}
SPL {X  -162.820, Y  +387.033, Z    +0.000, E1    -4.758, E3 +244144.255}
SPL {X  -162.820, Y  +390.967, Z    +0.000, E1    -9.918, E3 +244144.700}
SPL {X  -162.820, Y  +395.392, Z    +0.000, E1   -16.726, E3 +244143.141}
SPL {X  -162.820, Y  +402.654, Z    +0.000, E1   -26.492, E3 +244145.032}
SPL {X  -162.820, Y  +417.515, Z    +0.000, E1   -44.878, E3 +244144.149}
SPL {X  -162.820, Y  +462.065, Z    +0.000, E1   -61.507, E3 +244161.109}
SPL {X  -162.820, Y  +504.602, Z    +0.000, E1   -64.286, E3 +244186.635}
SPL {X  -162.820, Y  +539.530, Z    +0.000, E1   -60.821, E3 +244237.326}
ENDSPLINE

SPLINE
SPL {X  -162.820, Y  +534.172, Z    +0.000, E1   -58.470, E3 +244246.826}
ENDSPLINE

SPLINE
SPL {X  -162.820, Y  +543.678, Z    +0.000, E1   -58.515, E3 +244258.703}
SPL {X  -162.820, Y  +553.725, Z    +0.000, E1   -58.454, E3 +244271.964}
SPL {X  -162.820, Y  +562.850, Z    +0.000, E1   -58.373, E3 +244284.126}
SPL {X  -162.820, Y  +573.452, Z    +0.000, E1   -58.444, E3 +244297.339}
SPL {X  -162.820, Y  +583.632, Z    +0.000, E1   -58.444, E3 +244310.266}
SPL {X  -162.820, Y  +591.768, Z    +0.000, E1   -58.375, E3 +244321.130}
SPL {X  -162.820, Y  +601.090, Z    +0.000, E1   -58.519, E3 +244332.117}
SPL {X  -162.820, Y  +609.492, Z    +0.000, E1   -58.431, E3 +244343.422}
SPL {X  -162.820, Y  +617.241, Z    +0.000, E1   -58.340, E3 +244353.947}
SPL {X  -162.820, Y  +626.506, Z    +0.000, E1   -58.420, E3 +244365.329}
SPL {X  -162.820, Y  +635.919, Z    +0.000, E1   -58.604, E3 +244376.073}
SPL {X  -162.820, Y  +643.895, Z    +0.000, E1   -58.380, E3 +244387.838}
SPL {X  -162.820, Y  +653.118, Z    +0.000, E1   -58.401, E3 +244399.435}
SPL {X  -162.820, Y  +660.924, Z    +0.000, E1   -58.393, E3 +244409.503}
SPL {X  -162.820, Y  +670.459, Z    +0.000, E1   -58.489, E3 +244421.104}
SPL {X  -162.713, Y  +679.396, Z    +0.000, E1   -58.414, E3 +244433.003}
SPL {X  -162.301, Y  +686.495, Z    +0.000, E1   -58.302, E3 +244442.787}
SPL {X  -161.571, Y  +693.631, Z    +0.000, E1   -58.186, E3 +244452.751}
SPL {X  -160.411, Y  +701.402, Z    +0.000, E1   -58.100, E3 +244463.227}
SPL {X  -159.229, Y  +707.508, Z    +0.000, E1   -57.870, E3 +244472.465}
SPL {X  -157.825, Y  +713.519, Z    +0.000, E1   -57.630, E3 +244481.701}
SPL {X  -156.079, Y  +719.864, Z    +0.000, E1   -57.324, E3 +244491.664}
SPL {X  -154.064, Y  +726.175, Z    +0.000, E1   -57.042, E3 +244501.426}
SPL {X  -152.053, Y  +731.726, Z    +0.000, E1   -56.648, E3 +244510.711}
SPL {X  -150.108, Y  +736.570, Z    +0.000, E1   -56.283, E3 +244518.950}
SPL {X  -147.726, Y  +741.964, Z    +0.000, E1   -55.884, E3 +244527.986}
SPL {X  -145.163, Y  +747.242, Z    +0.000, E1   -55.517, E3 +244536.582}
SPL {X  -142.489, Y  +752.286, Z    +0.000, E1   -55.227, E3 +244544.409}
SPL {X  -136.074, Y  +762.910, Z    +0.000, E1   -57.336, E3 +244547.531}
SPL {X  -116.561, Y  +787.183, Z    +0.000, E1   -51.088, E3 +244631.999}
ENDSPLINE

SPLINE
SPL {X  -119.623, Y  +783.957, Z    +0.000, E1   -49.202, E3 +244756.532}
SPL {X  -149.958, Y  +736.927, Z    +0.000, E1   -34.772, E3 +244754.249}
SPL {X  -158.826, Y  +709.343, Z    +0.000, E1   -23.029, E3 +244762.592}
SPL {X  -161.344, Y  +695.370, Z    +0.000, E1   -15.607, E3 +244764.991}
SPL {X  -162.477, Y  +684.065, Z    +0.000, E1    -8.887, E3 +244764.621}
SPL {X  -162.776, Y  +677.290, Z    +0.000, E1    -4.406, E3 +244765.293}
SPL {X  -162.820, Y  +673.886, Z    +0.000, E1    -1.998, E3 +244765.121}
SPL {X  -162.820, Y  +670.901, Z    +0.000, E1    +0.338, E3 +244764.555}
SPL {X  -162.820, Y  +667.984, Z    +0.000, E1    +3.594, E3 +244764.387}
SPL {X  -162.820, Y  +664.667, Z    +0.000, E1    +7.867, E3 +244764.100}
SPL {X  -162.820, Y  +660.022, Z    +0.000, E1   +14.535, E3 +244763.997}
SPL {X  -162.820, Y  +653.408, Z    +0.000, E1   +24.221, E3 +244764.307}
SPL {X  -162.820, Y  +640.244, Z    +0.000, E1   +41.042, E3 +244764.351}
SPL {X  -162.820, Y  +592.517, Z    +0.000, E1   +60.575, E3 +244783.482}
SPL {X  -162.820, Y  +515.613, Z    +0.000, E1   +60.751, E3 +244857.317}
ENDSPLINE

SPLINE
SPL {X  -162.820, Y  +518.198, Z    +0.000, E1   +58.338, E3 +244870.473}
ENDSPLINE

SPLINE
SPL {X  -162.820, Y  +508.314, Z    +0.000, E1   +58.337, E3 +244883.169}
SPL {X  -162.820, Y  +498.518, Z    +0.000, E1   +58.346, E3 +244895.675}
SPL {X  -162.820, Y  +489.418, Z    +0.000, E1   +58.357, E3 +244907.265}
SPL {X  -162.820, Y  +479.904, Z    +0.000, E1   +58.389, E3 +244919.312}
SPL {X  -162.820, Y  +472.095, Z    +0.000, E1   +58.202, E3 +244930.492}
SPL {X  -162.820, Y  +463.661, Z    +0.000, E1   +58.370, E3 +244940.278}
SPL {X  -162.820, Y  +454.904, Z    +0.000, E1   +58.380, E3 +244951.444}
SPL {X  -162.820, Y  +446.206, Z    +0.000, E1   +58.278, E3 +244963.335}
SPL {X  -162.820, Y  +436.416, Z    +0.000, E1   +58.325, E3 +244975.575}
SPL {X  -162.820, Y  +426.628, Z    +0.000, E1   +58.432, E3 +244987.443}
SPL {X  -162.820, Y  +418.389, Z    +0.000, E1   +58.300, E3 +244998.846}
SPL {X  -162.820, Y  +412.292, Z    +0.000, E1   +58.070, E3 +245008.214}
SPL {X  -162.820, Y  +403.663, Z    +0.000, E1   +58.258, E3 +245018.154}
SPL {X  -162.820, Y  +397.157, Z    +0.000, E1   +58.054, E3 +245027.890}
SPL {X  -162.820, Y  +387.359, Z    +0.000, E1   +58.365, E3 +245038.519}
SPL {X  -162.810, Y  +378.731, Z    +0.000, E1   +58.366, E3 +245049.577}
SPL {X  -162.546, Y  +371.051, Z    +0.000, E1   +58.239, E3 +245060.297}
SPL {X  -161.863, Y  +362.875, Z    +0.000, E1   +58.273, E3 +245070.522}
SPL {X  -161.159, Y  +357.301, Z    +0.000, E1   +57.946, E3 +245079.822}
SPL {X  -159.864, Y  +349.614, Z    +0.000, E1   +57.922, E3 +245089.898}
SPL {X  -158.548, Y  +343.449, Z    +0.000, E1   +57.711, E3 +245099.072}
SPL {X  -156.580, Y  +335.856, Z    +0.000, E1   +57.340, E3 +245111.295}
SPL {X  -154.237, Y  +328.333, Z    +0.000, E1   +56.930, E3 +245123.214}
SPL {X  -152.732, Y  +324.078, Z    +0.000, E1   +56.482, E3 +245131.219}
SPL {X  -150.609, Y  +318.634, Z    +0.000, E1   +56.366, E3 +245138.913}
SPL {X  -148.206, Y  +313.080, Z    +0.000, E1   +55.888, E3 +245148.625}
SPL {X  -145.956, Y  +308.339, Z    +0.000, E1   +55.380, E3 +245157.301}
SPL {X  -142.234, Y  +301.255, Z    +0.000, E1   +55.418, E3 +245166.175}
SPL {X  -134.491, Y  +288.726, Z    +0.000, E1   +57.448, E3 +245171.831}
SPL {X  -115.845, Y  +266.087, Z    +0.000, E1   +50.276, E3 +245268.442}
SPL {X  -114.083, Y  +264.330, Z    +0.000, E1   +49.123, E3 +245307.152}
ENDSPLINE

SPLINE
SPL {X  -149.622, Y  +316.285, Z    +0.000, E1   +35.036, E3 +245375.664}
SPL {X  -158.704, Y  +344.121, Z    +0.000, E1   +23.312, E3 +245385.537}
SPL {X  -161.701, Y  +361.440, Z    +0.000, E1   +13.961, E3 +245384.608}
SPL {X  -162.691, Y  +374.019, Z    +0.000, E1    +6.263, E3 +245385.261}
SPL {X  -162.820, Y  +380.238, Z    +0.000, E1    +1.925, E3 +245384.945}
SPL {X  -162.820, Y  +383.454, Z    +0.000, E1    -0.619, E3 +245384.551}
SPL {X  -162.820, Y  +387.033, Z    +0.000, E1    -4.758, E3 +245384.255}
SPL {X  -162.820, Y  +390.967, Z    +0.000, E1    -9.918, E3 +245384.700}
SPL {X  -162.820, Y  +397.718, Z    +0.000, E1   -19.761, E3 +245384.074}
SPL {X  -162.820, Y  +405.058, Z    +0.000, E1   -29.962, E3 +245384.987}
SPL {X  -162.820, Y  +417.515, Z    +0.000, E1   -44.878, E3 +245384.149}
SPL {X  -162.820, Y  +462.065, Z    +0.000, E1   -61.507, E3 +245401.109}
SPL {X  -162.820, Y  +504.602, Z    +0.000, E1   -64.286, E3 +245426.635}
SPL {X  -162.820, Y  +539.530, Z    +0.000, E1   -60.821, E3 +245477.326}
ENDSPLINE

SPLINE
SPL {X  -162.820, Y  +534.172, Z    +0.000, E1   -58.470, E3 +245486.826}
ENDSPLINE

SPLINE
SPL {X  -162.820, Y  +543.678, Z    +0.000, E1   -58.515, E3 +245498.703}
SPL {X  -162.820, Y  +553.725, Z    +0.000, E1   -58.454, E3 +245511.964}
SPL {X  -162.820, Y  +562.850, Z    +0.000, E1   -58.373, E3 +245524.126}
SPL {X  -162.820, Y  +573.452, Z    +0.000, E1   -58.444, E3 +245537.339}
SPL {X  -162.820, Y  +583.632, Z    +0.000, E1   -58.444, E3 +245550.266}
SPL {X  -162.820, Y  +591.768, Z    +0.000, E1   -58.375, E3 +245561.130}
SPL {X  -162.820, Y  +601.090, Z    +0.000, E1   -58.519, E3 +245572.117}
SPL {X  -162.820, Y  +609.492, Z    +0.000, E1   -58.431, E3 +245583.422}
SPL {X  -162.820, Y  +617.241, Z    +0.000, E1   -58.340, E3 +245593.947}
SPL {X  -162.820, Y  +626.506, Z    +0.000, E1   -58.420, E3 +245605.329}
SPL {X  -162.820, Y  +635.919, Z    +0.000, E1   -58.604, E3 +245616.073}
SPL {X  -162.820, Y  +643.895, Z    +0.000, E1   -58.380, E3 +245627.838}
SPL {X  -162.820, Y  +653.118, Z    +0.000, E1   -58.401, E3 +245639.435}
SPL {X  -162.820, Y  +660.924, Z    +0.000, E1   -58.393, E3 +245649.503}
SPL {X  -162.820, Y  +670.459, Z    +0.000, E1   -58.489, E3 +245661.104}
SPL {X  -162.713, Y  +679.396, Z    +0.000, E1   -58.414, E3 +245673.003}
SPL {X  -162.301, Y  +686.495, Z    +0.000, E1   -58.302, E3 +245682.787}
SPL {X  -161.571, Y  +693.631, Z    +0.000, E1   -58.186, E3 +245692.751}
SPL {X  -160.411, Y  +701.402, Z    +0.000, E1   -58.100, E3 +245703.227}
SPL {X  -159.229, Y  +707.508, Z    +0.000, E1   -57.870, E3 +245712.465}
SPL {X  -157.825, Y  +713.519, Z    +0.000, E1   -57.630, E3 +245721.701}
SPL {X  -156.079, Y  +719.864, Z    +0.000, E1   -57.324, E3 +245731.664}
SPL {X  -154.064, Y  +726.175, Z    +0.000, E1   -57.042, E3 +245741.426}
SPL {X  -152.053, Y  +731.726, Z    +0.000, E1   -56.648, E3 +245750.711}
SPL {X  -150.108, Y  +736.570, Z    +0.000, E1   -56.283, E3 +245758.950}
SPL {X  -147.726, Y  +741.964, Z    +0.000, E1   -55.884, E3 +245767.986}
SPL {X  -145.163, Y  +747.242, Z    +0.000, E1   -55.517, E3 +245776.582}
SPL {X  -142.489, Y  +752.286, Z    +0.000, E1   -55.227, E3 +245784.409}
SPL {X  -136.074, Y  +762.910, Z    +0.000, E1   -57.336, E3 +245787.531}
SPL {X  -116.561, Y  +787.183, Z    +0.000, E1   -51.088, E3 +245871.999}
ENDSPLINE

SPLINE
SPL {X  -119.623, Y  +783.957, Z    +0.000, E1   -49.202, E3 +245996.532}
SPL {X  -149.958, Y  +736.927, Z    +0.000, E1   -34.772, E3 +245994.249}
SPL {X  -158.826, Y  +709.343, Z    +0.000, E1   -23.029, E3 +246002.592}
SPL {X  -161.800, Y  +691.694, Z    +0.000, E1   -13.520, E3 +246004.886}
SPL {X  -162.711, Y  +679.444, Z    +0.000, E1    -5.922, E3 +246004.960}
SPL {X  -162.820, Y  +672.303, Z    +0.000, E1    -0.875, E3 +246004.825}
SPL {X  -162.820, Y  +669.030, Z    +0.000, E1    +2.242, E3 +246004.397}
SPL {X  -162.820, Y  +664.667, Z    +0.000, E1    +7.867, E3 +246004.100}
SPL {X  -162.820, Y  +660.022, Z    +0.000, E1   +14.535, E3 +246003.997}
SPL {X  -162.820, Y  +653.408, Z    +0.000, E1   +24.221, E3 +246004.307}
SPL {X  -162.820, Y  +640.244, Z    +0.000, E1   +41.042, E3 +246004.351}
SPL {X  -162.820, Y  +592.517, Z    +0.000, E1   +60.575, E3 +246023.482}
SPL {X  -162.820, Y  +515.613, Z    +0.000, E1   +60.751, E3 +246097.317}
ENDSPLINE

SPLINE
SPL {X  -162.820, Y  +518.198, Z    +0.000, E1   +58.338, E3 +246110.473}
ENDSPLINE

SPLINE
SPL {X  -162.820, Y  +508.314, Z    +0.000, E1   +58.337, E3 +246123.169}
SPL {X  -162.820, Y  +498.518, Z    +0.000, E1   +58.346, E3 +246135.675}
SPL {X  -162.820, Y  +489.418, Z    +0.000, E1   +58.357, E3 +246147.265}
SPL {X  -162.820, Y  +479.904, Z    +0.000, E1   +58.389, E3 +246159.312}
SPL {X  -162.820, Y  +472.095, Z    +0.000, E1   +58.202, E3 +246170.492}
SPL {X  -162.820, Y  +463.661, Z    +0.000, E1   +58.370, E3 +246180.278}
SPL {X  -162.820, Y  +454.904, Z    +0.000, E1   +58.380, E3 +246191.444}
SPL {X  -162.820, Y  +446.206, Z    +0.000, E1   +58.278, E3 +246203.335}
SPL {X  -162.820, Y  +436.416, Z    +0.000, E1   +58.325, E3 +246215.575}
SPL {X  -162.820, Y  +426.628, Z    +0.000, E1   +58.432, E3 +246227.443}
SPL {X  -162.820, Y  +415.377, Z    +0.000, E1   +58.239, E3 +246243.375}
SPL {X  -162.820, Y  +403.663, Z    +0.000, E1   +58.258, E3 +246258.154}
SPL {X  -162.820, Y  +397.157, Z    +0.000, E1   +58.054, E3 +246267.890}
SPL {X  -162.820, Y  +387.359, Z    +0.000, E1   +58.365, E3 +246278.519}
SPL {X  -162.810, Y  +378.731, Z    +0.000, E1   +58.366, E3 +246289.577}
SPL {X  -162.546, Y  +371.051, Z    +0.000, E1   +58.239, E3 +246300.297}
SPL {X  -161.863, Y  +362.875, Z    +0.000, E1   +58.273, E3 +246310.522}
SPL {X  -161.159, Y  +357.301, Z    +0.000, E1   +57.946, E3 +246319.822}
SPL {X  -159.864, Y  +349.614, Z    +0.000, E1   +57.922, E3 +246329.898}
SPL {X  -158.548, Y  +343.449, Z    +0.000, E1   +57.711, E3 +246339.072}
SPL {X  -156.580, Y  +335.856, Z    +0.000, E1   +57.340, E3 +246351.295}
SPL {X  -154.237, Y  +328.333, Z    +0.000, E1   +56.930, E3 +246363.214}
SPL {X  -152.732, Y  +324.078, Z    +0.000, E1   +56.482, E3 +246371.219}
SPL {X  -150.609, Y  +318.634, Z    +0.000, E1   +56.366, E3 +246378.913}
SPL {X  -148.206, Y  +313.080, Z    +0.000, E1   +55.888, E3 +246388.625}
SPL {X  -145.956, Y  +308.339, Z    +0.000, E1   +55.380, E3 +246397.301}
SPL {X  -142.234, Y  +301.255, Z    +0.000, E1   +55.418, E3 +246406.175}
SPL {X  -134.491, Y  +288.726, Z    +0.000, E1   +57.448, E3 +246411.831}
SPL {X  -115.845, Y  +266.087, Z    +0.000, E1   +50.276, E3 +246508.442}
SPL {X  -114.083, Y  +264.330, Z    +0.000, E1   +49.123, E3 +246547.152}
ENDSPLINE

SPLINE
SPL {X  -136.188, Y  +291.263, Z    +0.000, E1   +45.457, E3 +246643.218}
SPL {X  -151.738, Y  +321.457, Z    +0.000, E1   +32.773, E3 +246610.387}
SPL {X  -158.704, Y  +344.121, Z    +0.000, E1   +23.312, E3 +246625.537}
SPL {X  -162.109, Y  +365.304, Z    +0.000, E1   +11.761, E3 +246624.839}
SPL {X  -162.811, Y  +378.776, Z    +0.000, E1    +3.078, E3 +246625.083}
SPL {X  -162.820, Y  +382.545, Z    +0.000, E1    +0.100, E3 +246624.644}
SPL {X  -162.820, Y  +384.317, Z    +0.000, E1    -1.618, E3 +246624.463}
SPL {X  -162.820, Y  +387.033, Z    +0.000, E1    -4.758, E3 +246624.255}
SPL {X  -162.820, Y  +390.967, Z    +0.000, E1    -9.918, E3 +246624.700}
SPL {X  -162.820, Y  +395.392, Z    +0.000, E1   -16.726, E3 +246623.141}
SPL {X  -162.820, Y  +402.654, Z    +0.000, E1   -26.492, E3 +246625.032}
SPL {X  -162.820, Y  +417.515, Z    +0.000, E1   -44.878, E3 +246624.149}
SPL {X  -162.820, Y  +462.065, Z    +0.000, E1   -61.507, E3 +246641.109}
SPL {X  -162.820, Y  +504.602, Z    +0.000, E1   -64.286, E3 +246666.635}
SPL {X  -162.820, Y  +535.709, Z    +0.000, E1   -59.182, E3 +246724.314}
SPL {X  -162.820, Y  +543.678, Z    +0.000, E1   -58.515, E3 +246738.703}
SPL {X  -162.820, Y  +553.725, Z    +0.000, E1   -58.454, E3 +246751.964}
SPL {X  -162.820, Y  +562.850, Z    +0.000, E1   -58.373, E3 +246764.126}
SPL {X  -162.820, Y  +573.452, Z    +0.000, E1   -58.444, E3 +246777.339}
SPL {X  -162.820, Y  +583.632, Z    +0.000, E1   -58.444, E3 +246790.266}
SPL {X  -162.820, Y  +591.768, Z    +0.000, E1   -58.375, E3 +246801.130}
SPL {X  -162.820, Y  +601.090, Z    +0.000, E1   -58.519, E3 +246812.117}
SPL {X  -162.820, Y  +609.492, Z    +0.000, E1   -58.431, E3 +246823.422}
SPL {X  -162.820, Y  +617.241, Z    +0.000, E1   -58.340, E3 +246833.947}
SPL {X  -162.820, Y  +626.506, Z    +0.000, E1   -58.420, E3 +246845.329}
SPL {X  -162.820, Y  +638.850, Z    +0.000, E1   -58.527, E3 +246860.545}
SPL {X  -162.820, Y  +651.112, Z    +0.000, E1   -58.411, E3 +246876.903}
SPL {X  -162.820, Y  +660.924, Z    +0.000, E1   -58.393, E3 +246889.503}
SPL {X  -162.820, Y  +670.459, Z    +0.000, E1   -58.489, E3 +246901.104}
SPL {X  -162.713, Y  +679.396, Z    +0.000, E1   -58.414, E3 +246913.003}
SPL {X  -162.301, Y  +686.495, Z    +0.000, E1   -58.302, E3 +246922.787}
SPL {X  -161.571, Y  +693.631, Z    +0.000, E1   -58.186, E3 +246932.751}
SPL {X  -160.411, Y  +701.402, Z    +0.000, E1   -58.100, E3 +246943.227}
SPL {X  -159.229, Y  +707.508, Z    +0.000, E1   -57.870, E3 +246952.465}
SPL {X  -157.825, Y  +713.519, Z    +0.000, E1   -57.630, E3 +246961.701}
SPL {X  -156.079, Y  +719.864, Z    +0.000, E1   -57.324, E3 +246971.664}
SPL {X  -154.064, Y  +726.175, Z    +0.000, E1   -57.042, E3 +246981.426}
SPL {X  -152.053, Y  +731.726, Z    +0.000, E1   -56.648, E3 +246990.711}
SPL {X  -150.108, Y  +736.570, Z    +0.000, E1   -56.283, E3 +246998.950}
SPL {X  -147.726, Y  +741.964, Z    +0.000, E1   -55.884, E3 +247007.986}
SPL {X  -145.163, Y  +747.242, Z    +0.000, E1   -55.517, E3 +247016.582}
SPL {X  -142.489, Y  +752.286, Z    +0.000, E1   -55.227, E3 +247024.409}
SPL {X  -136.074, Y  +762.910, Z    +0.000, E1   -57.336, E3 +247027.531}
SPL {X  -116.561, Y  +787.183, Z    +0.000, E1   -51.088, E3 +247111.999}
ENDSPLINE

SPLINE
SPL {X  -119.623, Y  +783.957, Z    +0.000, E1   -49.202, E3 +247236.532}
SPL {X  -149.958, Y  +736.927, Z    +0.000, E1   -34.772, E3 +247234.249}
SPL {X  -158.826, Y  +709.343, Z    +0.000, E1   -23.029, E3 +247242.592}
SPL {X  -161.344, Y  +695.370, Z    +0.000, E1   -15.607, E3 +247244.991}
SPL {X  -162.477, Y  +684.065, Z    +0.000, E1    -8.887, E3 +247244.621}
SPL {X  -162.776, Y  +677.290, Z    +0.000, E1    -4.406, E3 +247245.293}
SPL {X  -162.820, Y  +673.886, Z    +0.000, E1    -1.998, E3 +247245.121}
SPL {X  -162.820, Y  +670.901, Z    +0.000, E1    +0.338, E3 +247244.555}
SPL {X  -162.820, Y  +667.984, Z    +0.000, E1    +3.594, E3 +247244.387}
SPL {X  -162.820, Y  +664.667, Z    +0.000, E1    +7.867, E3 +247244.100}
SPL {X  -162.820, Y  +660.022, Z    +0.000, E1   +14.535, E3 +247243.997}
SPL {X  -162.820, Y  +653.408, Z    +0.000, E1   +24.221, E3 +247244.307}
SPL {X  -162.820, Y  +640.244, Z    +0.000, E1   +41.042, E3 +247244.351}
SPL {X  -162.820, Y  +592.517, Z    +0.000, E1   +60.575, E3 +247263.482}
SPL {X  -162.820, Y  +515.613, Z    +0.000, E1   +60.751, E3 +247337.317}
ENDSPLINE

SPLINE
SPL {X  -162.820, Y  +518.198, Z    +0.000, E1   +58.338, E3 +247350.473}
ENDSPLINE

SPLINE
SPL {X  -162.820, Y  +508.314, Z    +0.000, E1   +58.337, E3 +247363.169}
SPL {X  -162.820, Y  +498.518, Z    +0.000, E1   +58.346, E3 +247375.675}
SPL {X  -162.820, Y  +489.418, Z    +0.000, E1   +58.357, E3 +247387.265}
SPL {X  -162.820, Y  +479.904, Z    +0.000, E1   +58.389, E3 +247399.312}
SPL {X  -162.820, Y  +472.095, Z    +0.000, E1   +58.202, E3 +247410.492}
SPL {X  -162.820, Y  +463.661, Z    +0.000, E1   +58.370, E3 +247420.278}
SPL {X  -162.820, Y  +454.904, Z    +0.000, E1   +58.380, E3 +247431.444}
SPL {X  -162.820, Y  +446.206, Z    +0.000, E1   +58.278, E3 +247443.335}
SPL {X  -162.820, Y  +436.416, Z    +0.000, E1   +58.325, E3 +247455.575}
SPL {X  -162.820, Y  +426.628, Z    +0.000, E1   +58.432, E3 +247467.443}
SPL {X  -162.820, Y  +415.377, Z    +0.000, E1   +58.239, E3 +247483.375}
SPL {X  -162.820, Y  +403.663, Z    +0.000, E1   +58.258, E3 +247498.154}
SPL {X  -162.820, Y  +397.157, Z    +0.000, E1   +58.054, E3 +247507.890}
SPL {X  -162.820, Y  +387.359, Z    +0.000, E1   +58.365, E3 +247518.519}
SPL {X  -162.810, Y  +378.731, Z    +0.000, E1   +58.366, E3 +247529.577}
SPL {X  -162.546, Y  +371.051, Z    +0.000, E1   +58.239, E3 +247540.297}
SPL {X  -161.863, Y  +362.875, Z    +0.000, E1   +58.273, E3 +247550.522}
SPL {X  -161.159, Y  +357.301, Z    +0.000, E1   +57.946, E3 +247559.822}
SPL {X  -159.864, Y  +349.614, Z    +0.000, E1   +57.922, E3 +247569.898}
SPL {X  -158.300, Y  +342.404, Z    +0.000, E1   +57.579, E3 +247581.344}
SPL {X  -156.187, Y  +334.499, Z    +0.000, E1   +57.331, E3 +247593.004}
SPL {X  -154.237, Y  +328.333, Z    +0.000, E1   +56.930, E3 +247603.214}
SPL {X  -152.732, Y  +324.078, Z    +0.000, E1   +56.482, E3 +247611.219}
SPL {X  -150.609, Y  +318.634, Z    +0.000, E1   +56.366, E3 +247618.913}
SPL {X  -148.206, Y  +313.080, Z    +0.000, E1   +55.888, E3 +247628.625}
SPL {X  -145.956, Y  +308.339, Z    +0.000, E1   +55.380, E3 +247637.301}
SPL {X  -143.330, Y  +303.254, Z    +0.000, E1   +55.057, E3 +247645.421}
SPL {X  -137.431, Y  +293.190, Z    +0.000, E1   +56.809, E3 +247649.584}
SPL {X  -115.845, Y  +266.087, Z    +0.000, E1   +50.276, E3 +247748.442}
SPL {X  -114.083, Y  +264.330, Z    +0.000, E1   +49.123, E3 +247787.152}
ENDSPLINE

SPLINE
SPL {X  -149.622, Y  +316.285, Z    +0.000, E1   +35.036, E3 +247855.664}
SPL {X  -158.704, Y  +344.121, Z    +0.000, E1   +23.312, E3 +247865.537}
SPL {X  -162.109, Y  +365.304, Z    +0.000, E1   +11.761, E3 +247864.839}
SPL {X  -162.811, Y  +378.776, Z    +0.000, E1    +3.078, E3 +247865.083}
SPL {X  -162.820, Y  +383.454, Z    +0.000, E1    -0.619, E3 +247864.551}
SPL {X  -162.820, Y  +387.033, Z    +0.000, E1    -4.758, E3 +247864.255}
SPL {X  -162.820, Y  +390.967, Z    +0.000, E1    -9.918, E3 +247864.700}
SPL {X  -162.820, Y  +397.718, Z    +0.000, E1   -19.761, E3 +247864.074}
SPL {X  -162.820, Y  +405.058, Z    +0.000, E1   -29.962, E3 +247864.987}
SPL {X  -162.820, Y  +417.515, Z    +0.000, E1   -44.878, E3 +247864.149}
SPL {X  -162.820, Y  +462.065, Z    +0.000, E1   -61.507, E3 +247881.109}
SPL {X  -162.820, Y  +504.602, Z    +0.000, E1   -64.286, E3 +247906.635}
SPL {X  -162.820, Y  +535.709, Z    +0.000, E1   -59.182, E3 +247964.314}
SPL {X  -162.820, Y  +543.678, Z    +0.000, E1   -58.515, E3 +247978.703}
SPL {X  -162.820, Y  +553.725, Z    +0.000, E1   -58.454, E3 +247991.964}
SPL {X  -162.820, Y  +562.850, Z    +0.000, E1   -58.373, E3 +248004.126}
SPL {X  -162.820, Y  +571.217, Z    +0.000, E1   -58.397, E3 +248014.679}
SPL {X  -162.820, Y  +581.879, Z    +0.000, E1   -58.475, E3 +248027.932}
SPL {X  -162.820, Y  +591.768, Z    +0.000, E1   -58.375, E3 +248041.130}
SPL {X  -162.820, Y  +601.090, Z    +0.000, E1   -58.519, E3 +248052.117}
SPL {X  -162.820, Y  +609.492, Z    +0.000, E1   -58.431, E3 +248063.422}
SPL {X  -162.820, Y  +617.241, Z    +0.000, E1   -58.340, E3 +248073.947}
SPL {X  -162.820, Y  +626.506, Z    +0.000, E1   -58.420, E3 +248085.329}
SPL {X  -162.820, Y  +638.850, Z    +0.000, E1   -58.527, E3 +248100.545}
SPL {X  -162.820, Y  +651.112, Z    +0.000, E1   -58.411, E3 +248116.903}
SPL {X  -162.820, Y  +660.924, Z    +0.000, E1   -58.393, E3 +248129.503}
SPL {X  -162.820, Y  +670.459, Z    +0.000, E1   -58.489, E3 +248141.104}
SPL {X  -162.713, Y  +679.396, Z    +0.000, E1   -58.414, E3 +248153.003}
SPL {X  -162.301, Y  +686.495, Z    +0.000, E1   -58.302, E3 +248162.787}
SPL {X  -161.571, Y  +693.631, Z    +0.000, E1   -58.186, E3 +248172.751}
SPL {X  -160.411, Y  +701.402, Z    +0.000, E1   -58.100, E3 +248183.227}
SPL {X  -159.229, Y  +707.508, Z    +0.000, E1   -57.870, E3 +248192.465}
SPL {X  -157.825, Y  +713.519, Z    +0.000, E1   -57.630, E3 +248201.701}
SPL {X  -156.079, Y  +719.864, Z    +0.000, E1   -57.324, E3 +248211.664}
SPL {X  -154.064, Y  +726.175, Z    +0.000, E1   -57.042, E3 +248221.426}
SPL {X  -152.053, Y  +731.726, Z    +0.000, E1   -56.648, E3 +248230.711}
SPL {X  -150.108, Y  +736.570, Z    +0.000, E1   -56.283, E3 +248238.950}
SPL {X  -147.726, Y  +741.964, Z    +0.000, E1   -55.884, E3 +248247.986}
SPL {X  -145.163, Y  +747.242, Z    +0.000, E1   -55.517, E3 +248256.582}
SPL {X  -142.489, Y  +752.286, Z    +0.000, E1   -55.227, E3 +248264.409}
SPL {X  -136.074, Y  +762.910, Z    +0.000, E1   -57.336, E3 +248267.531}
SPL {X  -116.561, Y  +787.183, Z    +0.000, E1   -51.088, E3 +248351.999}
ENDSPLINE

SPLINE
SPL {X  -119.623, Y  +783.957, Z    +0.000, E1   -49.202, E3 +248476.532}
SPL {X  -149.958, Y  +736.927, Z    +0.000, E1   -34.772, E3 +248474.249}
SPL {X  -158.826, Y  +709.343, Z    +0.000, E1   -23.029, E3 +248482.592}
SPL {X  -161.344, Y  +695.370, Z    +0.000, E1   -15.607, E3 +248484.991}
SPL {X  -162.477, Y  +684.065, Z    +0.000, E1    -8.887, E3 +248484.621}
SPL {X  -162.813, Y  +675.055, Z    +0.000, E1    -2.911, E3 +248485.184}
SPL {X  -162.820, Y  +670.901, Z    +0.000, E1    +0.338, E3 +248484.555}
SPL {X  -162.820, Y  +667.984, Z    +0.000, E1    +3.594, E3 +248484.387}
SPL {X  -162.820, Y  +664.667, Z    +0.000, E1    +7.867, E3 +248484.100}
SPL {X  -162.820, Y  +660.022, Z    +0.000, E1   +14.535, E3 +248483.997}
SPL {X  -162.820, Y  +653.408, Z    +0.000, E1   +24.221, E3 +248484.307}
SPL {X  -162.820, Y  +640.244, Z    +0.000, E1   +41.042, E3 +248484.351}
SPL {X  -162.820, Y  +592.517, Z    +0.000, E1   +60.575, E3 +248503.482}
SPL {X  -162.820, Y  +515.613, Z    +0.000, E1   +60.751, E3 +248577.317}
ENDSPLINE

SPLINE
SPL {X  -162.820, Y  +518.198, Z    +0.000, E1   +58.338, E3 +248590.473}
ENDSPLINE

SPLINE
SPL {X  -162.820, Y  +508.314, Z    +0.000, E1   +58.337, E3 +248603.169}
SPL {X  -162.820, Y  +498.518, Z    +0.000, E1   +58.346, E3 +248615.675}
SPL {X  -162.820, Y  +489.418, Z    +0.000, E1   +58.357, E3 +248627.265}
SPL {X  -162.820, Y  +479.904, Z    +0.000, E1   +58.389, E3 +248639.312}
SPL {X  -162.820, Y  +472.095, Z    +0.000, E1   +58.202, E3 +248650.492}
SPL {X  -162.820, Y  +463.661, Z    +0.000, E1   +58.370, E3 +248660.278}
SPL {X  -162.820, Y  +454.904, Z    +0.000, E1   +58.380, E3 +248671.444}
SPL {X  -162.820, Y  +446.206, Z    +0.000, E1   +58.278, E3 +248683.335}
SPL {X  -162.820, Y  +436.416, Z    +0.000, E1   +58.325, E3 +248695.575}
SPL {X  -162.820, Y  +426.628, Z    +0.000, E1   +58.432, E3 +248707.443}
SPL {X  -162.820, Y  +418.389, Z    +0.000, E1   +58.300, E3 +248718.846}
SPL {X  -162.820, Y  +412.292, Z    +0.000, E1   +58.070, E3 +248728.214}
SPL {X  -162.820, Y  +403.663, Z    +0.000, E1   +58.258, E3 +248738.154}
SPL {X  -162.820, Y  +397.157, Z    +0.000, E1   +58.054, E3 +248747.890}
SPL {X  -162.820, Y  +387.359, Z    +0.000, E1   +58.365, E3 +248758.519}
SPL {X  -162.810, Y  +378.731, Z    +0.000, E1   +58.366, E3 +248769.577}
SPL {X  -162.546, Y  +371.051, Z    +0.000, E1   +58.239, E3 +248780.297}
SPL {X  -161.863, Y  +362.875, Z    +0.000, E1   +58.273, E3 +248790.522}
SPL {X  -161.159, Y  +357.301, Z    +0.000, E1   +57.946, E3 +248799.822}
SPL {X  -159.864, Y  +349.614, Z    +0.000, E1   +57.922, E3 +248809.898}
SPL {X  -158.300, Y  +342.404, Z    +0.000, E1   +57.579, E3 +248821.344}
SPL {X  -156.187, Y  +334.499, Z    +0.000, E1   +57.331, E3 +248833.004}
SPL {X  -154.237, Y  +328.333, Z    +0.000, E1   +56.930, E3 +248843.214}
SPL {X  -152.732, Y  +324.078, Z    +0.000, E1   +56.482, E3 +248851.219}
SPL {X  -150.609, Y  +318.634, Z    +0.000, E1   +56.366, E3 +248858.913}
SPL {X  -148.206, Y  +313.080, Z    +0.000, E1   +55.888, E3 +248868.625}
SPL {X  -145.956, Y  +308.339, Z    +0.000, E1   +55.380, E3 +248877.301}
SPL {X  -143.330, Y  +303.254, Z    +0.000, E1   +55.057, E3 +248885.421}
SPL {X  -137.431, Y  +293.190, Z    +0.000, E1   +56.809, E3 +248889.584}
SPL {X  -115.845, Y  +266.087, Z    +0.000, E1   +50.276, E3 +248988.442}
SPL {X  -114.083, Y  +264.330, Z    +0.000, E1   +49.123, E3 +249027.152}
ENDSPLINE

SPLINE
SPL {X  -149.622, Y  +316.285, Z    +0.000, E1   +35.036, E3 +249095.664}
SPL {X  -158.704, Y  +344.121, Z    +0.000, E1   +23.312, E3 +249105.537}
SPL {X  -161.701, Y  +361.440, Z    +0.000, E1   +13.961, E3 +249104.608}
SPL {X  -162.691, Y  +374.019, Z    +0.000, E1    +6.263, E3 +249105.261}
SPL {X  -162.820, Y  +380.238, Z    +0.000, E1    +1.925, E3 +249104.945}
SPL {X  -162.820, Y  +383.454, Z    +0.000, E1    -0.619, E3 +249104.551}
SPL {X  -162.820, Y  +387.033, Z    +0.000, E1    -4.758, E3 +249104.255}
SPL {X  -162.820, Y  +390.967, Z    +0.000, E1    -9.918, E3 +249104.700}
SPL {X  -162.820, Y  +395.392, Z    +0.000, E1   -16.726, E3 +249103.141}
SPL {X  -162.820, Y  +402.654, Z    +0.000, E1   -26.492, E3 +249105.032}
SPL {X  -162.820, Y  +417.515, Z    +0.000, E1   -44.878, E3 +249104.149}
SPL {X  -162.820, Y  +462.065, Z    +0.000, E1   -61.507, E3 +249121.109}
SPL {X  -162.820, Y  +504.602, Z    +0.000, E1   -64.286, E3 +249146.635}
SPL {X  -162.820, Y  +535.709, Z    +0.000, E1   -59.182, E3 +249204.314}
SPL {X  -162.820, Y  +543.678, Z    +0.000, E1   -58.515, E3 +249218.703}
SPL {X  -162.820, Y  +553.725, Z    +0.000, E1   -58.454, E3 +249231.964}
SPL {X  -162.820, Y  +562.850, Z    +0.000, E1   -58.373, E3 +249244.126}
SPL {X  -162.820, Y  +573.452, Z    +0.000, E1   -58.444, E3 +249257.339}
SPL {X  -162.820, Y  +583.632, Z    +0.000, E1   -58.444, E3 +249270.266}
SPL {X  -162.820, Y  +591.768, Z    +0.000, E1   -58.375, E3 +249281.130}
SPL {X  -162.820, Y  +601.090, Z    +0.000, E1   -58.519, E3 +249292.117}
SPL {X  -162.820, Y  +609.492, Z    +0.000, E1   -58.431, E3 +249303.422}
SPL {X  -162.820, Y  +617.241, Z    +0.000, E1   -58.340, E3 +249313.947}
SPL {X  -162.820, Y  +626.506, Z    +0.000, E1   -58.420, E3 +249325.329}
SPL {X  -162.820, Y  +635.919, Z    +0.000, E1   -58.604, E3 +249336.073}
SPL {X  -162.820, Y  +643.895, Z    +0.000, E1   -58.380, E3 +249347.838}
SPL {X  -162.820, Y  +653.118, Z    +0.000, E1   -58.401, E3 +249359.435}
SPL {X  -162.820, Y  +660.924, Z    +0.000, E1   -58.393, E3 +249369.503}
SPL {X  -162.820, Y  +670.459, Z    +0.000, E1   -58.489, E3 +249381.104}
SPL {X  -162.713, Y  +679.396, Z    +0.000, E1   -58.414, E3 +249393.003}
SPL {X  -162.301, Y  +686.495, Z    +0.000, E1   -58.302, E3 +249402.787}
SPL {X  -161.571, Y  +693.631, Z    +0.000, E1   -58.186, E3 +249412.751}
SPL {X  -160.411, Y  +701.402, Z    +0.000, E1   -58.100, E3 +249423.227}
SPL {X  -159.229, Y  +707.508, Z    +0.000, E1   -57.870, E3 +249432.465}
SPL {X  -157.825, Y  +713.519, Z    +0.000, E1   -57.630, E3 +249441.701}
SPL {X  -156.079, Y  +719.864, Z    +0.000, E1   -57.324, E3 +249451.664}
SPL {X  -154.064, Y  +726.175, Z    +0.000, E1   -57.042, E3 +249461.426}
SPL {X  -152.053, Y  +731.726, Z    +0.000, E1   -56.648, E3 +249470.711}
SPL {X  -150.108, Y  +736.570, Z    +0.000, E1   -56.283, E3 +249478.950}
SPL {X  -147.726, Y  +741.964, Z    +0.000, E1   -55.884, E3 +249487.986}
SPL {X  -145.163, Y  +747.242, Z    +0.000, E1   -55.517, E3 +249496.582}
SPL {X  -142.489, Y  +752.286, Z    +0.000, E1   -55.227, E3 +249504.409}
SPL {X  -136.074, Y  +762.910, Z    +0.000, E1   -57.336, E3 +249507.531}
SPL {X  -121.244, Y  +782.175, Z    +0.000, E1   -51.023, E3 +249579.476}
SPL {X  -114.422, Y  +789.335, Z    +0.000, E1   -51.094, E3 +249598.092}
ENDSPLINE

SPLINE
SPL {X  -119.623, Y  +783.957, Z    +0.000, E1   -49.202, E3 +249716.532}
SPL {X  -149.958, Y  +736.927, Z    +0.000, E1   -34.772, E3 +249714.249}
SPL {X  -158.826, Y  +709.343, Z    +0.000, E1   -23.029, E3 +249722.592}
SPL {X  -161.800, Y  +691.694, Z    +0.000, E1   -13.520, E3 +249724.886}
SPL {X  -162.711, Y  +679.444, Z    +0.000, E1    -5.922, E3 +249724.960}
SPL {X  -162.820, Y  +672.303, Z    +0.000, E1    -0.875, E3 +249724.825}
SPL {X  -162.820, Y  +669.030, Z    +0.000, E1    +2.242, E3 +249724.397}
SPL {X  -162.820, Y  +664.667, Z    +0.000, E1    +7.867, E3 +249724.100}
SPL {X  -162.820, Y  +660.022, Z    +0.000, E1   +14.535, E3 +249723.997}
SPL {X  -162.820, Y  +653.408, Z    +0.000, E1   +24.221, E3 +249724.307}
SPL {X  -162.820, Y  +640.244, Z    +0.000, E1   +41.042, E3 +249724.351}
SPL {X  -162.820, Y  +592.517, Z    +0.000, E1   +60.575, E3 +249743.482}
SPL {X  -162.820, Y  +515.613, Z    +0.000, E1   +60.751, E3 +249817.317}
ENDSPLINE

SPLINE
SPL {X  -162.820, Y  +518.198, Z    +0.000, E1   +58.338, E3 +249830.473}
ENDSPLINE

SPLINE
SPL {X  -162.820, Y  +508.314, Z    +0.000, E1   +58.337, E3 +249843.169}
SPL {X  -162.820, Y  +498.518, Z    +0.000, E1   +58.346, E3 +249855.675}
SPL {X  -162.820, Y  +489.418, Z    +0.000, E1   +58.357, E3 +249867.265}
SPL {X  -162.820, Y  +479.904, Z    +0.000, E1   +58.389, E3 +249879.312}
SPL {X  -162.820, Y  +472.095, Z    +0.000, E1   +58.202, E3 +249890.492}
SPL {X  -162.820, Y  +463.661, Z    +0.000, E1   +58.370, E3 +249900.278}
SPL {X  -162.820, Y  +454.904, Z    +0.000, E1   +58.380, E3 +249911.444}
SPL {X  -162.820, Y  +446.206, Z    +0.000, E1   +58.278, E3 +249923.335}
SPL {X  -162.820, Y  +436.416, Z    +0.000, E1   +58.325, E3 +249935.575}
SPL {X  -162.820, Y  +426.628, Z    +0.000, E1   +58.432, E3 +249947.443}
SPL {X  -162.820, Y  +415.377, Z    +0.000, E1   +58.239, E3 +249963.375}
SPL {X  -162.820, Y  +403.663, Z    +0.000, E1   +58.258, E3 +249978.154}
SPL {X  -162.820, Y  +397.157, Z    +0.000, E1   +58.054, E3 +249987.890}
SPL {X  -162.820, Y  +387.359, Z    +0.000, E1   +58.365, E3 +249998.519}
SPL {X  -162.810, Y  +378.731, Z    +0.000, E1   +58.366, E3 +250009.577}
SPL {X  -162.546, Y  +371.051, Z    +0.000, E1   +58.239, E3 +250020.297}
SPL {X  -161.863, Y  +362.875, Z    +0.000, E1   +58.273, E3 +250030.522}
SPL {X  -161.159, Y  +357.301, Z    +0.000, E1   +57.946, E3 +250039.822}
SPL {X  -159.864, Y  +349.614, Z    +0.000, E1   +57.922, E3 +250049.898}
SPL {X  -158.300, Y  +342.404, Z    +0.000, E1   +57.579, E3 +250061.344}
SPL {X  -156.187, Y  +334.499, Z    +0.000, E1   +57.331, E3 +250073.004}
SPL {X  -154.237, Y  +328.333, Z    +0.000, E1   +56.930, E3 +250083.214}
SPL {X  -152.732, Y  +324.078, Z    +0.000, E1   +56.482, E3 +250091.219}
SPL {X  -150.609, Y  +318.634, Z    +0.000, E1   +56.366, E3 +250098.913}
SPL {X  -148.206, Y  +313.080, Z    +0.000, E1   +55.888, E3 +250108.625}
SPL {X  -145.956, Y  +308.339, Z    +0.000, E1   +55.380, E3 +250117.301}
SPL {X  -143.330, Y  +303.254, Z    +0.000, E1   +55.057, E3 +250125.421}
SPL {X  -137.431, Y  +293.190, Z    +0.000, E1   +56.809, E3 +250129.584}
SPL {X  -115.845, Y  +266.087, Z    +0.000, E1   +50.276, E3 +250228.442}
SPL {X  -114.083, Y  +264.330, Z    +0.000, E1   +49.123, E3 +250267.152}
ENDSPLINE

SPLINE
SPL {X  -149.622, Y  +316.285, Z    +0.000, E1   +35.036, E3 +250335.664}
SPL {X  -158.704, Y  +344.121, Z    +0.000, E1   +23.312, E3 +250345.537}
SPL {X  -162.109, Y  +365.304, Z    +0.000, E1   +11.761, E3 +250344.839}
SPL {X  -162.811, Y  +378.776, Z    +0.000, E1    +3.078, E3 +250345.083}
SPL {X  -162.820, Y  +382.545, Z    +0.000, E1    +0.100, E3 +250344.644}
SPL {X  -162.820, Y  +384.317, Z    +0.000, E1    -1.618, E3 +250344.463}
SPL {X  -162.820, Y  +387.033, Z    +0.000, E1    -4.758, E3 +250344.255}
SPL {X  -162.820, Y  +390.967, Z    +0.000, E1    -9.918, E3 +250344.700}
SPL {X  -162.820, Y  +395.392, Z    +0.000, E1   -16.726, E3 +250343.141}
SPL {X  -162.820, Y  +402.654, Z    +0.000, E1   -26.492, E3 +250345.032}
SPL {X  -162.820, Y  +417.515, Z    +0.000, E1   -44.878, E3 +250344.149}
SPL {X  -162.820, Y  +462.065, Z    +0.000, E1   -61.507, E3 +250361.109}
SPL {X  -162.820, Y  +504.602, Z    +0.000, E1   -64.286, E3 +250386.635}
SPL {X  -162.820, Y  +539.530, Z    +0.000, E1   -60.821, E3 +250437.326}
ENDSPLINE

SPLINE
SPL {X  -162.820, Y  +534.172, Z    +0.000, E1   -58.470, E3 +250446.826}
ENDSPLINE

SPLINE
SPL {X  -162.820, Y  +543.678, Z    +0.000, E1   -58.515, E3 +250458.703}
SPL {X  -162.820, Y  +553.725, Z    +0.000, E1   -58.454, E3 +250471.964}
SPL {X  -162.820, Y  +562.850, Z    +0.000, E1   -58.373, E3 +250484.126}
SPL {X  -162.820, Y  +573.452, Z    +0.000, E1   -58.444, E3 +250497.339}
SPL {X  -162.820, Y  +583.632, Z    +0.000, E1   -58.444, E3 +250510.266}
SPL {X  -162.820, Y  +591.768, Z    +0.000, E1   -58.375, E3 +250521.130}
SPL {X  -162.820, Y  +601.090, Z    +0.000, E1   -58.519, E3 +250532.117}
SPL {X  -162.820, Y  +609.492, Z    +0.000, E1   -58.431, E3 +250543.422}
SPL {X  -162.820, Y  +617.241, Z    +0.000, E1   -58.340, E3 +250553.947}
SPL {X  -162.820, Y  +626.506, Z    +0.000, E1   -58.420, E3 +250565.329}
SPL {X  -162.820, Y  +635.919, Z    +0.000, E1   -58.604, E3 +250576.073}
SPL {X  -162.820, Y  +643.895, Z    +0.000, E1   -58.380, E3 +250587.838}
SPL {X  -162.820, Y  +653.118, Z    +0.000, E1   -58.401, E3 +250599.435}
SPL {X  -162.820, Y  +660.924, Z    +0.000, E1   -58.393, E3 +250609.503}
SPL {X  -162.820, Y  +670.459, Z    +0.000, E1   -58.489, E3 +250621.104}
SPL {X  -162.713, Y  +679.396, Z    +0.000, E1   -58.414, E3 +250633.003}
SPL {X  -162.301, Y  +686.495, Z    +0.000, E1   -58.302, E3 +250642.787}
SPL {X  -161.571, Y  +693.631, Z    +0.000, E1   -58.186, E3 +250652.751}
SPL {X  -160.411, Y  +701.402, Z    +0.000, E1   -58.100, E3 +250663.227}
SPL {X  -159.229, Y  +707.508, Z    +0.000, E1   -57.870, E3 +250672.465}
SPL {X  -157.825, Y  +713.519, Z    +0.000, E1   -57.630, E3 +250681.701}
SPL {X  -156.079, Y  +719.864, Z    +0.000, E1   -57.324, E3 +250691.664}
SPL {X  -154.064, Y  +726.175, Z    +0.000, E1   -57.042, E3 +250701.426}
SPL {X  -152.053, Y  +731.726, Z    +0.000, E1   -56.648, E3 +250710.711}
SPL {X  -150.108, Y  +736.570, Z    +0.000, E1   -56.283, E3 +250718.950}
SPL {X  -147.726, Y  +741.964, Z    +0.000, E1   -55.884, E3 +250727.986}
SPL {X  -145.163, Y  +747.242, Z    +0.000, E1   -55.517, E3 +250736.582}
SPL {X  -142.489, Y  +752.286, Z    +0.000, E1   -55.227, E3 +250744.409}
SPL {X  -136.074, Y  +762.910, Z    +0.000, E1   -57.336, E3 +250747.531}
SPL {X  -116.561, Y  +787.183, Z    +0.000, E1   -51.088, E3 +250831.999}
ENDSPLINE

SPLINE
SPL {X  -119.623, Y  +783.957, Z    +0.000, E1   -49.202, E3 +250956.532}
SPL {X  -149.958, Y  +736.927, Z    +0.000, E1   -34.772, E3 +250954.249}
SPL {X  -158.826, Y  +709.343, Z    +0.000, E1   -23.029, E3 +250962.592}
SPL {X  -161.344, Y  +695.370, Z    +0.000, E1   -15.607, E3 +250964.991}
SPL {X  -162.477, Y  +684.065, Z    +0.000, E1    -8.887, E3 +250964.621}
SPL {X  -162.776, Y  +677.290, Z    +0.000, E1    -4.406, E3 +250965.293}
SPL {X  -162.820, Y  +673.886, Z    +0.000, E1    -1.998, E3 +250965.121}
SPL {X  -162.820, Y  +670.901, Z    +0.000, E1    +0.338, E3 +250964.555}
SPL {X  -162.820, Y  +667.984, Z    +0.000, E1    +3.594, E3 +250964.387}
SPL {X  -162.820, Y  +664.667, Z    +0.000, E1    +7.867, E3 +250964.100}
SPL {X  -162.820, Y  +660.022, Z    +0.000, E1   +14.535, E3 +250963.997}
SPL {X  -162.820, Y  +653.408, Z    +0.000, E1   +24.221, E3 +250964.307}
SPL {X  -162.820, Y  +640.244, Z    +0.000, E1   +41.042, E3 +250964.351}
SPL {X  -162.820, Y  +592.517, Z    +0.000, E1   +60.575, E3 +250983.482}
SPL {X  -162.820, Y  +515.613, Z    +0.000, E1   +60.751, E3 +251057.317}
ENDSPLINE

SPLINE
SPL {X  -162.820, Y  +518.198, Z    +0.000, E1   +58.338, E3 +251070.473}
ENDSPLINE

SPLINE
SPL {X  -162.820, Y  +508.314, Z    +0.000, E1   +58.337, E3 +251083.169}
SPL {X  -162.820, Y  +498.518, Z    +0.000, E1   +58.346, E3 +251095.675}
SPL {X  -162.820, Y  +487.033, Z    +0.000, E1   +58.385, E3 +251110.273}
SPL {X  -162.820, Y  +474.470, Z    +0.000, E1   +58.318, E3 +251126.839}
SPL {X  -162.820, Y  +463.661, Z    +0.000, E1   +58.370, E3 +251140.278}
SPL {X  -162.820, Y  +454.904, Z    +0.000, E1   +58.380, E3 +251151.444}
SPL {X  -162.820, Y  +446.206, Z    +0.000, E1   +58.278, E3 +251163.335}
SPL {X  -162.820, Y  +436.416, Z    +0.000, E1   +58.325, E3 +251175.575}
SPL {X  -162.820, Y  +426.628, Z    +0.000, E1   +58.432, E3 +251187.443}
SPL {X  -162.820, Y  +415.377, Z    +0.000, E1   +58.239, E3 +251203.375}
SPL {X  -162.820, Y  +403.663, Z    +0.000, E1   +58.258, E3 +251218.154}
SPL {X  -162.820, Y  +397.157, Z    +0.000, E1   +58.054, E3 +251227.890}
SPL {X  -162.820, Y  +387.359, Z    +0.000, E1   +58.365, E3 +251238.519}
SPL {X  -162.810, Y  +378.731, Z    +0.000, E1   +58.366, E3 +251249.577}
SPL {X  -162.546, Y  +371.051, Z    +0.000, E1   +58.239, E3 +251260.297}
SPL {X  -161.863, Y  +362.875, Z    +0.000, E1   +58.273, E3 +251270.522}
SPL {X  -161.159, Y  +357.301, Z    +0.000, E1   +57.946, E3 +251279.822}
SPL {X  -159.864, Y  +349.614, Z    +0.000, E1   +57.922, E3 +251289.898}
SPL {X  -158.548, Y  +343.449, Z    +0.000, E1   +57.711, E3 +251299.072}
SPL {X  -156.580, Y  +335.856, Z    +0.000, E1   +57.340, E3 +251311.295}
SPL {X  -154.237, Y  +328.333, Z    +0.000, E1   +56.930, E3 +251323.214}
SPL {X  -152.732, Y  +324.078, Z    +0.000, E1   +56.482, E3 +251331.219}
SPL {X  -150.609, Y  +318.634, Z    +0.000, E1   +56.366, E3 +251338.913}
SPL {X  -148.206, Y  +313.080, Z    +0.000, E1   +55.888, E3 +251348.625}
SPL {X  -145.956, Y  +308.339, Z    +0.000, E1   +55.380, E3 +251357.301}
SPL {X  -143.330, Y  +303.254, Z    +0.000, E1   +55.057, E3 +251365.421}
SPL {X  -137.431, Y  +293.190, Z    +0.000, E1   +56.809, E3 +251369.584}
SPL {X  -115.845, Y  +266.087, Z    +0.000, E1   +50.276, E3 +251468.442}
SPL {X  -114.083, Y  +264.330, Z    +0.000, E1   +49.123, E3 +251507.152}
ENDSPLINE

SPLINE
SPL {X  -149.622, Y  +316.285, Z    +0.000, E1   +35.036, E3 +251575.664}
SPL {X  -158.704, Y  +344.121, Z    +0.000, E1   +23.312, E3 +251585.537}
SPL {X  -161.701, Y  +361.440, Z    +0.000, E1   +13.961, E3 +251584.608}
SPL {X  -162.691, Y  +374.019, Z    +0.000, E1    +6.263, E3 +251585.261}
SPL {X  -162.820, Y  +380.238, Z    +0.000, E1    +1.925, E3 +251584.945}
SPL {X  -162.820, Y  +383.454, Z    +0.000, E1    -0.619, E3 +251584.551}
SPL {X  -162.820, Y  +387.033, Z    +0.000, E1    -4.758, E3 +251584.255}
SPL {X  -162.820, Y  +390.967, Z    +0.000, E1    -9.918, E3 +251584.700}
SPL {X  -162.820, Y  +397.718, Z    +0.000, E1   -19.761, E3 +251584.074}
SPL {X  -162.820, Y  +405.058, Z    +0.000, E1   -29.962, E3 +251584.987}
SPL {X  -162.820, Y  +417.515, Z    +0.000, E1   -44.878, E3 +251584.149}
SPL {X  -162.820, Y  +462.065, Z    +0.000, E1   -61.507, E3 +251601.109}
SPL {X  -162.820, Y  +504.602, Z    +0.000, E1   -64.286, E3 +251626.635}
SPL {X  -162.820, Y  +535.709, Z    +0.000, E1   -59.182, E3 +251684.314}
SPL {X  -162.820, Y  +543.678, Z    +0.000, E1   -58.515, E3 +251698.703}
SPL {X  -162.820, Y  +553.725, Z    +0.000, E1   -58.454, E3 +251711.964}
SPL {X  -162.820, Y  +562.850, Z    +0.000, E1   -58.373, E3 +251724.126}
SPL {X  -162.820, Y  +573.452, Z    +0.000, E1   -58.444, E3 +251737.339}
SPL {X  -162.820, Y  +583.632, Z    +0.000, E1   -58.444, E3 +251750.266}
SPL {X  -162.820, Y  +591.768, Z    +0.000, E1   -58.375, E3 +251761.130}
SPL {X  -162.820, Y  +601.090, Z    +0.000, E1   -58.519, E3 +251772.117}
SPL {X  -162.820, Y  +609.492, Z    +0.000, E1   -58.431, E3 +251783.422}
SPL {X  -162.820, Y  +617.241, Z    +0.000, E1   -58.340, E3 +251793.947}
SPL {X  -162.820, Y  +626.506, Z    +0.000, E1   -58.420, E3 +251805.329}
SPL {X  -162.820, Y  +635.919, Z    +0.000, E1   -58.604, E3 +251816.073}
SPL {X  -162.820, Y  +643.895, Z    +0.000, E1   -58.380, E3 +251827.838}
SPL {X  -162.820, Y  +653.118, Z    +0.000, E1   -58.401, E3 +251839.435}
SPL {X  -162.820, Y  +660.924, Z    +0.000, E1   -58.393, E3 +251849.503}
SPL {X  -162.820, Y  +670.459, Z    +0.000, E1   -58.489, E3 +251861.104}
SPL {X  -162.713, Y  +679.396, Z    +0.000, E1   -58.414, E3 +251873.003}
SPL {X  -162.301, Y  +686.495, Z    +0.000, E1   -58.302, E3 +251882.787}
SPL {X  -161.571, Y  +693.631, Z    +0.000, E1   -58.186, E3 +251892.751}
SPL {X  -160.411, Y  +701.402, Z    +0.000, E1   -58.100, E3 +251903.227}
SPL {X  -159.229, Y  +707.508, Z    +0.000, E1   -57.870, E3 +251912.465}
SPL {X  -157.825, Y  +713.519, Z    +0.000, E1   -57.630, E3 +251921.701}
SPL {X  -156.079, Y  +719.864, Z    +0.000, E1   -57.324, E3 +251931.664}
SPL {X  -154.064, Y  +726.175, Z    +0.000, E1   -57.042, E3 +251941.426}
SPL {X  -152.053, Y  +731.726, Z    +0.000, E1   -56.648, E3 +251950.711}
SPL {X  -150.108, Y  +736.570, Z    +0.000, E1   -56.283, E3 +251958.950}
SPL {X  -147.726, Y  +741.964, Z    +0.000, E1   -55.884, E3 +251967.986}
SPL {X  -145.163, Y  +747.242, Z    +0.000, E1   -55.517, E3 +251976.582}
SPL {X  -142.489, Y  +752.286, Z    +0.000, E1   -55.227, E3 +251984.409}
SPL {X  -136.074, Y  +762.910, Z    +0.000, E1   -57.336, E3 +251987.531}
SPL {X  -116.561, Y  +787.183, Z    +0.000, E1   -51.088, E3 +252071.999}
ENDSPLINE

SPLINE
SPL {X  -119.623, Y  +783.957, Z    +0.000, E1   -49.202, E3 +252196.532}
SPL {X  -149.958, Y  +736.927, Z    +0.000, E1   -34.772, E3 +252194.249}
SPL {X  -158.826, Y  +709.343, Z    +0.000, E1   -23.029, E3 +252202.592}
SPL {X  -161.344, Y  +695.370, Z    +0.000, E1   -15.607, E3 +252204.991}
SPL {X  -162.477, Y  +684.065, Z    +0.000, E1    -8.887, E3 +252204.621}
SPL {X  -162.776, Y  +677.290, Z    +0.000, E1    -4.406, E3 +252205.293}
SPL {X  -162.820, Y  +672.303, Z    +0.000, E1    -0.875, E3 +252204.825}
SPL {X  -162.820, Y  +669.030, Z    +0.000, E1    +2.242, E3 +252204.397}
SPL {X  -162.820, Y  +664.667, Z    +0.000, E1    +7.867, E3 +252204.100}
SPL {X  -162.820, Y  +660.022, Z    +0.000, E1   +14.535, E3 +252203.997}
SPL {X  -162.820, Y  +653.408, Z    +0.000, E1   +24.221, E3 +252204.307}
SPL {X  -162.820, Y  +640.244, Z    +0.000, E1   +41.042, E3 +252204.351}
SPL {X  -162.820, Y  +592.517, Z    +0.000, E1   +60.575, E3 +252223.482}
SPL {X  -162.820, Y  +515.613, Z    +0.000, E1   +60.751, E3 +252297.317}
ENDSPLINE

SPLINE
SPL {X  -162.820, Y  +518.198, Z    +0.000, E1   +58.338, E3 +252310.473}
ENDSPLINE

SPLINE
SPL {X  -162.820, Y  +508.314, Z    +0.000, E1   +58.337, E3 +252323.169}
SPL {X  -162.820, Y  +498.518, Z    +0.000, E1   +58.346, E3 +252335.675}
SPL {X  -162.820, Y  +487.033, Z    +0.000, E1   +58.385, E3 +252350.273}
SPL {X  -162.820, Y  +474.470, Z    +0.000, E1   +58.318, E3 +252366.839}
SPL {X  -162.820, Y  +463.661, Z    +0.000, E1   +58.370, E3 +252380.278}
SPL {X  -162.820, Y  +454.904, Z    +0.000, E1   +58.380, E3 +252391.444}
SPL {X  -162.820, Y  +446.206, Z    +0.000, E1   +58.278, E3 +252403.335}
SPL {X  -162.820, Y  +436.416, Z    +0.000, E1   +58.325, E3 +252415.575}
SPL {X  -162.820, Y  +426.628, Z    +0.000, E1   +58.432, E3 +252427.443}
SPL {X  -162.820, Y  +415.377, Z    +0.000, E1   +58.239, E3 +252443.375}
SPL {X  -162.820, Y  +403.663, Z    +0.000, E1   +58.258, E3 +252458.154}
SPL {X  -162.820, Y  +397.157, Z    +0.000, E1   +58.054, E3 +252467.890}
SPL {X  -162.820, Y  +387.359, Z    +0.000, E1   +58.365, E3 +252478.519}
SPL {X  -162.810, Y  +378.731, Z    +0.000, E1   +58.366, E3 +252489.577}
SPL {X  -162.546, Y  +371.051, Z    +0.000, E1   +58.239, E3 +252500.297}
SPL {X  -161.863, Y  +362.875, Z    +0.000, E1   +58.273, E3 +252510.522}
SPL {X  -161.159, Y  +357.301, Z    +0.000, E1   +57.946, E3 +252519.822}
SPL {X  -159.864, Y  +349.614, Z    +0.000, E1   +57.922, E3 +252529.898}
SPL {X  -158.300, Y  +342.404, Z    +0.000, E1   +57.579, E3 +252541.344}
SPL {X  -156.187, Y  +334.499, Z    +0.000, E1   +57.331, E3 +252553.004}
SPL {X  -154.237, Y  +328.333, Z    +0.000, E1   +56.930, E3 +252563.214}
SPL {X  -152.732, Y  +324.078, Z    +0.000, E1   +56.482, E3 +252571.219}
SPL {X  -150.609, Y  +318.634, Z    +0.000, E1   +56.366, E3 +252578.913}
SPL {X  -148.206, Y  +313.080, Z    +0.000, E1   +55.888, E3 +252588.625}
SPL {X  -145.956, Y  +308.339, Z    +0.000, E1   +55.380, E3 +252597.301}
SPL {X  -143.330, Y  +303.254, Z    +0.000, E1   +55.057, E3 +252605.421}
SPL {X  -137.431, Y  +293.190, Z    +0.000, E1   +56.809, E3 +252609.584}
SPL {X  -115.845, Y  +266.087, Z    +0.000, E1   +50.276, E3 +252708.442}
SPL {X  -114.083, Y  +264.330, Z    +0.000, E1   +49.123, E3 +252747.152}
ENDSPLINE

SPLINE
SPL {X  -149.622, Y  +316.285, Z    +0.000, E1   +35.036, E3 +252815.664}
SPL {X  -158.704, Y  +344.121, Z    +0.000, E1   +23.312, E3 +252825.537}
SPL {X  -161.701, Y  +361.440, Z    +0.000, E1   +13.961, E3 +252824.608}
SPL {X  -162.691, Y  +374.019, Z    +0.000, E1    +6.263, E3 +252825.261}
SPL {X  -162.820, Y  +380.238, Z    +0.000, E1    +1.925, E3 +252824.945}
SPL {X  -162.820, Y  +383.454, Z    +0.000, E1    -0.619, E3 +252824.551}
SPL {X  -162.820, Y  +387.033, Z    +0.000, E1    -4.758, E3 +252824.255}
SPL {X  -162.820, Y  +390.967, Z    +0.000, E1    -9.918, E3 +252824.700}
SPL {X  -162.820, Y  +395.392, Z    +0.000, E1   -16.726, E3 +252823.141}
SPL {X  -162.820, Y  +402.654, Z    +0.000, E1   -26.492, E3 +252825.032}
SPL {X  -162.820, Y  +417.515, Z    +0.000, E1   -44.878, E3 +252824.149}
SPL {X  -162.820, Y  +462.065, Z    +0.000, E1   -61.507, E3 +252841.109}
SPL {X  -162.820, Y  +504.602, Z    +0.000, E1   -64.286, E3 +252866.635}
SPL {X  -162.820, Y  +535.709, Z    +0.000, E1   -59.182, E3 +252924.314}
SPL {X  -162.820, Y  +543.678, Z    +0.000, E1   -58.515, E3 +252938.703}
SPL {X  -162.820, Y  +553.725, Z    +0.000, E1   -58.454, E3 +252951.964}
SPL {X  -162.820, Y  +562.850, Z    +0.000, E1   -58.373, E3 +252964.126}
SPL {X  -162.820, Y  +573.452, Z    +0.000, E1   -58.444, E3 +252977.339}
SPL {X  -162.820, Y  +583.632, Z    +0.000, E1   -58.444, E3 +252990.266}
SPL {X  -162.820, Y  +591.768, Z    +0.000, E1   -58.375, E3 +253001.130}
SPL {X  -162.820, Y  +601.090, Z    +0.000, E1   -58.519, E3 +253012.117}
SPL {X  -162.820, Y  +609.492, Z    +0.000, E1   -58.431, E3 +253023.422}
SPL {X  -162.820, Y  +617.241, Z    +0.000, E1   -58.340, E3 +253033.947}
SPL {X  -162.820, Y  +626.506, Z    +0.000, E1   -58.420, E3 +253045.329}
SPL {X  -162.820, Y  +638.850, Z    +0.000, E1   -58.527, E3 +253060.545}
SPL {X  -162.820, Y  +651.112, Z    +0.000, E1   -58.411, E3 +253076.903}
SPL {X  -162.820, Y  +660.924, Z    +0.000, E1   -58.393, E3 +253089.503}
SPL {X  -162.820, Y  +670.459, Z    +0.000, E1   -58.489, E3 +253101.104}
SPL {X  -162.713, Y  +679.396, Z    +0.000, E1   -58.414, E3 +253113.003}
SPL {X  -162.301, Y  +686.495, Z    +0.000, E1   -58.302, E3 +253122.787}
SPL {X  -161.571, Y  +693.631, Z    +0.000, E1   -58.186, E3 +253132.751}
SPL {X  -160.411, Y  +701.402, Z    +0.000, E1   -58.100, E3 +253143.227}
SPL {X  -159.229, Y  +707.508, Z    +0.000, E1   -57.870, E3 +253152.465}
SPL {X  -157.825, Y  +713.519, Z    +0.000, E1   -57.630, E3 +253161.701}
SPL {X  -156.079, Y  +719.864, Z    +0.000, E1   -57.324, E3 +253171.664}
SPL {X  -154.064, Y  +726.175, Z    +0.000, E1   -57.042, E3 +253181.426}
SPL {X  -152.053, Y  +731.726, Z    +0.000, E1   -56.648, E3 +253190.711}
SPL {X  -150.108, Y  +736.570, Z    +0.000, E1   -56.283, E3 +253198.950}
SPL {X  -147.726, Y  +741.964, Z    +0.000, E1   -55.884, E3 +253207.986}
SPL {X  -145.163, Y  +747.242, Z    +0.000, E1   -55.517, E3 +253216.582}
SPL {X  -142.489, Y  +752.286, Z    +0.000, E1   -55.227, E3 +253224.409}
SPL {X  -136.074, Y  +762.910, Z    +0.000, E1   -57.336, E3 +253227.531}
SPL {X  -116.561, Y  +787.183, Z    +0.000, E1   -51.088, E3 +253311.999}
ENDSPLINE

SPLINE
SPL {X  -119.623, Y  +783.957, Z    +0.000, E1   -49.202, E3 +253436.532}
SPL {X  -149.958, Y  +736.927, Z    +0.000, E1   -34.772, E3 +253434.249}
SPL {X  -158.826, Y  +709.343, Z    +0.000, E1   -23.029, E3 +253442.592}
SPL {X  -161.800, Y  +691.694, Z    +0.000, E1   -13.520, E3 +253444.886}
SPL {X  -162.711, Y  +679.444, Z    +0.000, E1    -5.922, E3 +253444.960}
SPL {X  -162.820, Y  +673.886, Z    +0.000, E1    -1.998, E3 +253445.121}
SPL {X  -162.820, Y  +670.901, Z    +0.000, E1    +0.338, E3 +253444.555}
SPL {X  -162.820, Y  +667.984, Z    +0.000, E1    +3.594, E3 +253444.387}
SPL {X  -162.820, Y  +664.667, Z    +0.000, E1    +7.867, E3 +253444.100}
SPL {X  -162.820, Y  +660.022, Z    +0.000, E1   +14.535, E3 +253443.997}
SPL {X  -162.820, Y  +653.408, Z    +0.000, E1   +24.221, E3 +253444.307}
SPL {X  -162.820, Y  +640.244, Z    +0.000, E1   +41.042, E3 +253444.351}
SPL {X  -162.820, Y  +592.517, Z    +0.000, E1   +60.575, E3 +253463.482}
SPL {X  -162.820, Y  +515.613, Z    +0.000, E1   +60.751, E3 +253537.317}
ENDSPLINE

SPLINE
SPL {X  -162.820, Y  +518.198, Z    +0.000, E1   +58.338, E3 +253550.473}
ENDSPLINE

SPLINE
SPL {X  -162.820, Y  +508.314, Z    +0.000, E1   +58.337, E3 +253563.169}
SPL {X  -162.820, Y  +498.518, Z    +0.000, E1   +58.346, E3 +253575.675}
SPL {X  -162.820, Y  +489.418, Z    +0.000, E1   +58.357, E3 +253587.265}
SPL {X  -162.820, Y  +479.904, Z    +0.000, E1   +58.389, E3 +253599.312}
SPL {X  -162.820, Y  +472.095, Z    +0.000, E1   +58.202, E3 +253610.492}
SPL {X  -162.820, Y  +463.661, Z    +0.000, E1   +58.370, E3 +253620.278}
SPL {X  -162.820, Y  +454.904, Z    +0.000, E1   +58.380, E3 +253631.444}
SPL {X  -162.820, Y  +446.206, Z    +0.000, E1   +58.278, E3 +253643.335}
SPL {X  -162.820, Y  +436.416, Z    +0.000, E1   +58.325, E3 +253655.575}
SPL {X  -162.820, Y  +426.628, Z    +0.000, E1   +58.432, E3 +253667.443}
SPL {X  -162.820, Y  +415.377, Z    +0.000, E1   +58.239, E3 +253683.375}
SPL {X  -162.820, Y  +403.663, Z    +0.000, E1   +58.258, E3 +253698.154}
SPL {X  -162.820, Y  +397.157, Z    +0.000, E1   +58.054, E3 +253707.890}
SPL {X  -162.820, Y  +387.359, Z    +0.000, E1   +58.365, E3 +253718.519}
SPL {X  -162.810, Y  +378.731, Z    +0.000, E1   +58.366, E3 +253729.577}
SPL {X  -162.546, Y  +371.051, Z    +0.000, E1   +58.239, E3 +253740.297}
SPL {X  -161.863, Y  +362.875, Z    +0.000, E1   +58.273, E3 +253750.522}
SPL {X  -161.159, Y  +357.301, Z    +0.000, E1   +57.946, E3 +253759.822}
SPL {X  -159.864, Y  +349.614, Z    +0.000, E1   +57.922, E3 +253769.898}
SPL {X  -158.300, Y  +342.404, Z    +0.000, E1   +57.579, E3 +253781.344}
SPL {X  -156.187, Y  +334.499, Z    +0.000, E1   +57.331, E3 +253793.004}
SPL {X  -154.237, Y  +328.333, Z    +0.000, E1   +56.930, E3 +253803.214}
SPL {X  -152.732, Y  +324.078, Z    +0.000, E1   +56.482, E3 +253811.219}
SPL {X  -150.609, Y  +318.634, Z    +0.000, E1   +56.366, E3 +253818.913}
SPL {X  -148.206, Y  +313.080, Z    +0.000, E1   +55.888, E3 +253828.625}
SPL {X  -145.956, Y  +308.339, Z    +0.000, E1   +55.380, E3 +253837.301}
SPL {X  -142.234, Y  +301.255, Z    +0.000, E1   +55.418, E3 +253846.175}
SPL {X  -134.491, Y  +288.726, Z    +0.000, E1   +57.448, E3 +253851.831}
SPL {X  -115.845, Y  +266.087, Z    +0.000, E1   +50.276, E3 +253948.442}
SPL {X  -114.083, Y  +264.330, Z    +0.000, E1   +49.123, E3 +253987.152}
ENDSPLINE

SPLINE
SPL {X  -136.188, Y  +291.263, Z    +0.000, E1   +45.457, E3 +254083.218}
SPL {X  -151.738, Y  +321.457, Z    +0.000, E1   +32.773, E3 +254050.387}
SPL {X  -158.704, Y  +344.121, Z    +0.000, E1   +23.312, E3 +254065.537}
SPL {X  -161.701, Y  +361.440, Z    +0.000, E1   +13.961, E3 +254064.608}
SPL {X  -162.691, Y  +374.019, Z    +0.000, E1    +6.263, E3 +254065.261}
SPL {X  -162.820, Y  +380.238, Z    +0.000, E1    +1.925, E3 +254064.945}
SPL {X  -162.820, Y  +383.454, Z    +0.000, E1    -0.619, E3 +254064.551}
SPL {X  -162.820, Y  +387.033, Z    +0.000, E1    -4.758, E3 +254064.255}
SPL {X  -162.820, Y  +390.967, Z    +0.000, E1    -9.918, E3 +254064.700}
SPL {X  -162.820, Y  +395.392, Z    +0.000, E1   -16.726, E3 +254063.141}
SPL {X  -162.820, Y  +402.654, Z    +0.000, E1   -26.492, E3 +254065.032}
SPL {X  -162.820, Y  +417.515, Z    +0.000, E1   -44.878, E3 +254064.149}
SPL {X  -162.820, Y  +462.065, Z    +0.000, E1   -61.507, E3 +254081.109}
SPL {X  -162.820, Y  +504.602, Z    +0.000, E1   -64.286, E3 +254106.635}
SPL {X  -162.820, Y  +535.709, Z    +0.000, E1   -59.182, E3 +254164.314}
SPL {X  -162.820, Y  +543.678, Z    +0.000, E1   -58.515, E3 +254178.703}
SPL {X  -162.820, Y  +553.725, Z    +0.000, E1   -58.454, E3 +254191.964}
SPL {X  -162.820, Y  +562.850, Z    +0.000, E1   -58.373, E3 +254204.126}
SPL {X  -162.820, Y  +571.217, Z    +0.000, E1   -58.397, E3 +254214.679}
SPL {X  -162.820, Y  +581.879, Z    +0.000, E1   -58.475, E3 +254227.932}
SPL {X  -162.820, Y  +591.768, Z    +0.000, E1   -58.375, E3 +254241.130}
SPL {X  -162.820, Y  +601.090, Z    +0.000, E1   -58.519, E3 +254252.117}
SPL {X  -162.820, Y  +609.492, Z    +0.000, E1   -58.431, E3 +254263.422}
SPL {X  -162.820, Y  +617.241, Z    +0.000, E1   -58.340, E3 +254273.947}
SPL {X  -162.820, Y  +626.506, Z    +0.000, E1   -58.420, E3 +254285.329}
SPL {X  -162.820, Y  +638.850, Z    +0.000, E1   -58.527, E3 +254300.545}
SPL {X  -162.820, Y  +651.112, Z    +0.000, E1   -58.411, E3 +254316.903}
SPL {X  -162.820, Y  +660.924, Z    +0.000, E1   -58.393, E3 +254329.503}
SPL {X  -162.820, Y  +670.459, Z    +0.000, E1   -58.489, E3 +254341.104}
SPL {X  -162.713, Y  +679.396, Z    +0.000, E1   -58.414, E3 +254353.003}
SPL {X  -162.301, Y  +686.495, Z    +0.000, E1   -58.302, E3 +254362.787}
SPL {X  -161.571, Y  +693.631, Z    +0.000, E1   -58.186, E3 +254372.751}
SPL {X  -160.411, Y  +701.402, Z    +0.000, E1   -58.100, E3 +254383.227}
SPL {X  -159.229, Y  +707.508, Z    +0.000, E1   -57.870, E3 +254392.465}
SPL {X  -157.825, Y  +713.519, Z    +0.000, E1   -57.630, E3 +254401.701}
SPL {X  -156.079, Y  +719.864, Z    +0.000, E1   -57.324, E3 +254411.664}
SPL {X  -154.064, Y  +726.175, Z    +0.000, E1   -57.042, E3 +254421.426}
SPL {X  -152.053, Y  +731.726, Z    +0.000, E1   -56.648, E3 +254430.711}
SPL {X  -150.108, Y  +736.570, Z    +0.000, E1   -56.283, E3 +254438.950}
SPL {X  -147.726, Y  +741.964, Z    +0.000, E1   -55.884, E3 +254447.986}
SPL {X  -145.163, Y  +747.242, Z    +0.000, E1   -55.517, E3 +254456.582}
SPL {X  -142.489, Y  +752.286, Z    +0.000, E1   -55.227, E3 +254464.409}
SPL {X  -136.074, Y  +762.910, Z    +0.000, E1   -57.336, E3 +254467.531}
SPL {X  -116.561, Y  +787.183, Z    +0.000, E1   -51.088, E3 +254551.999}
ENDSPLINE

SPLINE
SPL {X  -119.623, Y  +783.957, Z    +0.000, E1   -49.202, E3 +254676.532}
SPL {X  -149.958, Y  +736.927, Z    +0.000, E1   -34.772, E3 +254674.249}
SPL {X  -158.826, Y  +709.343, Z    +0.000, E1   -23.029, E3 +254682.592}
SPL {X  -161.344, Y  +695.370, Z    +0.000, E1   -15.607, E3 +254684.991}
SPL {X  -162.477, Y  +684.065, Z    +0.000, E1    -8.887, E3 +254684.621}
SPL {X  -162.813, Y  +675.055, Z    +0.000, E1    -2.911, E3 +254685.184}
SPL {X  -162.820, Y  +670.901, Z    +0.000, E1    +0.338, E3 +254684.555}
SPL {X  -162.820, Y  +667.984, Z    +0.000, E1    +3.594, E3 +254684.387}
SPL {X  -162.820, Y  +664.667, Z    +0.000, E1    +7.867, E3 +254684.100}
SPL {X  -162.820, Y  +660.022, Z    +0.000, E1   +14.535, E3 +254683.997}
SPL {X  -162.820, Y  +653.408, Z    +0.000, E1   +24.221, E3 +254684.307}
SPL {X  -162.820, Y  +640.244, Z    +0.000, E1   +41.042, E3 +254684.351}
SPL {X  -162.820, Y  +592.517, Z    +0.000, E1   +60.575, E3 +254703.482}
SPL {X  -162.820, Y  +515.613, Z    +0.000, E1   +60.751, E3 +254777.317}
ENDSPLINE

SPLINE
SPL {X  -162.820, Y  +518.198, Z    +0.000, E1   +58.338, E3 +254790.473}
ENDSPLINE

SPLINE
SPL {X  -162.820, Y  +508.314, Z    +0.000, E1   +58.337, E3 +254803.169}
SPL {X  -162.820, Y  +498.518, Z    +0.000, E1   +58.346, E3 +254815.675}
SPL {X  -162.820, Y  +489.418, Z    +0.000, E1   +58.357, E3 +254827.265}
SPL {X  -162.820, Y  +479.904, Z    +0.000, E1   +58.389, E3 +254839.312}
SPL {X  -162.820, Y  +472.095, Z    +0.000, E1   +58.202, E3 +254850.492}
SPL {X  -162.820, Y  +463.661, Z    +0.000, E1   +58.370, E3 +254860.278}
SPL {X  -162.820, Y  +454.904, Z    +0.000, E1   +58.380, E3 +254871.444}
SPL {X  -162.820, Y  +446.206, Z    +0.000, E1   +58.278, E3 +254883.335}
SPL {X  -162.820, Y  +436.416, Z    +0.000, E1   +58.325, E3 +254895.575}
SPL {X  -162.820, Y  +426.628, Z    +0.000, E1   +58.432, E3 +254907.443}
SPL {X  -162.820, Y  +418.389, Z    +0.000, E1   +58.300, E3 +254918.846}
SPL {X  -162.820, Y  +412.292, Z    +0.000, E1   +58.070, E3 +254928.214}
SPL {X  -162.820, Y  +403.663, Z    +0.000, E1   +58.258, E3 +254938.154}
SPL {X  -162.820, Y  +397.157, Z    +0.000, E1   +58.054, E3 +254947.890}
SPL {X  -162.820, Y  +387.359, Z    +0.000, E1   +58.365, E3 +254958.519}
SPL {X  -162.810, Y  +378.731, Z    +0.000, E1   +58.366, E3 +254969.577}
SPL {X  -162.546, Y  +371.051, Z    +0.000, E1   +58.239, E3 +254980.297}
SPL {X  -161.863, Y  +362.875, Z    +0.000, E1   +58.273, E3 +254990.522}
SPL {X  -161.159, Y  +357.301, Z    +0.000, E1   +57.946, E3 +254999.822}
SPL {X  -159.864, Y  +349.614, Z    +0.000, E1   +57.922, E3 +255009.898}
SPL {X  -158.300, Y  +342.404, Z    +0.000, E1   +57.579, E3 +255021.344}
SPL {X  -156.187, Y  +334.499, Z    +0.000, E1   +57.331, E3 +255033.004}
SPL {X  -154.237, Y  +328.333, Z    +0.000, E1   +56.930, E3 +255043.214}
SPL {X  -152.732, Y  +324.078, Z    +0.000, E1   +56.482, E3 +255051.219}
SPL {X  -150.609, Y  +318.634, Z    +0.000, E1   +56.366, E3 +255058.913}
SPL {X  -148.206, Y  +313.080, Z    +0.000, E1   +55.888, E3 +255068.625}
SPL {X  -145.956, Y  +308.339, Z    +0.000, E1   +55.380, E3 +255077.301}
SPL {X  -143.330, Y  +303.254, Z    +0.000, E1   +55.057, E3 +255085.421}
SPL {X  -137.431, Y  +293.190, Z    +0.000, E1   +56.809, E3 +255089.584}
SPL {X  -115.845, Y  +266.087, Z    +0.000, E1   +50.276, E3 +255188.442}
SPL {X  -114.083, Y  +264.330, Z    +0.000, E1   +49.123, E3 +255227.152}
ENDSPLINE

SPLINE
SPL {X  -136.188, Y  +291.263, Z    +0.000, E1   +45.457, E3 +255323.218}
SPL {X  -151.738, Y  +321.457, Z    +0.000, E1   +32.773, E3 +255290.387}
SPL {X  -158.704, Y  +344.121, Z    +0.000, E1   +23.312, E3 +255305.537}
SPL {X  -161.701, Y  +361.440, Z    +0.000, E1   +13.961, E3 +255304.608}
SPL {X  -162.691, Y  +374.019, Z    +0.000, E1    +6.263, E3 +255305.261}
SPL {X  -162.820, Y  +380.238, Z    +0.000, E1    +1.925, E3 +255304.945}
SPL {X  -162.820, Y  +383.454, Z    +0.000, E1    -0.619, E3 +255304.551}
SPL {X  -162.820, Y  +387.033, Z    +0.000, E1    -4.758, E3 +255304.255}
SPL {X  -162.820, Y  +390.967, Z    +0.000, E1    -9.918, E3 +255304.700}
SPL {X  -162.820, Y  +397.718, Z    +0.000, E1   -19.761, E3 +255304.074}
SPL {X  -162.820, Y  +405.058, Z    +0.000, E1   -29.962, E3 +255304.987}
SPL {X  -162.820, Y  +417.515, Z    +0.000, E1   -44.878, E3 +255304.149}
SPL {X  -162.820, Y  +462.065, Z    +0.000, E1   -61.507, E3 +255321.109}
SPL {X  -162.820, Y  +504.602, Z    +0.000, E1   -64.286, E3 +255346.635}
SPL {X  -162.820, Y  +539.530, Z    +0.000, E1   -60.821, E3 +255397.326}
ENDSPLINE

SPLINE
SPL {X  -162.820, Y  +534.172, Z    +0.000, E1   -58.470, E3 +255406.826}
ENDSPLINE

SPLINE
SPL {X  -162.820, Y  +543.678, Z    +0.000, E1   -58.515, E3 +255418.703}
SPL {X  -162.820, Y  +553.725, Z    +0.000, E1   -58.454, E3 +255431.964}
SPL {X  -162.820, Y  +562.850, Z    +0.000, E1   -58.373, E3 +255444.126}
SPL {X  -162.820, Y  +573.452, Z    +0.000, E1   -58.444, E3 +255457.339}
SPL {X  -162.820, Y  +583.632, Z    +0.000, E1   -58.444, E3 +255470.266}
SPL {X  -162.820, Y  +591.768, Z    +0.000, E1   -58.375, E3 +255481.130}
SPL {X  -162.820, Y  +601.090, Z    +0.000, E1   -58.519, E3 +255492.117}
SPL {X  -162.820, Y  +609.492, Z    +0.000, E1   -58.431, E3 +255503.422}
SPL {X  -162.820, Y  +617.241, Z    +0.000, E1   -58.340, E3 +255513.947}
SPL {X  -162.820, Y  +626.506, Z    +0.000, E1   -58.420, E3 +255525.329}
SPL {X  -162.820, Y  +635.919, Z    +0.000, E1   -58.604, E3 +255536.073}
SPL {X  -162.820, Y  +643.895, Z    +0.000, E1   -58.380, E3 +255547.838}
SPL {X  -162.820, Y  +653.118, Z    +0.000, E1   -58.401, E3 +255559.435}
SPL {X  -162.820, Y  +660.924, Z    +0.000, E1   -58.393, E3 +255569.503}
SPL {X  -162.820, Y  +670.459, Z    +0.000, E1   -58.489, E3 +255581.104}
SPL {X  -162.713, Y  +679.396, Z    +0.000, E1   -58.414, E3 +255593.003}
SPL {X  -162.301, Y  +686.495, Z    +0.000, E1   -58.302, E3 +255602.787}
SPL {X  -161.571, Y  +693.631, Z    +0.000, E1   -58.186, E3 +255612.751}
SPL {X  -160.411, Y  +701.402, Z    +0.000, E1   -58.100, E3 +255623.227}
SPL {X  -159.229, Y  +707.508, Z    +0.000, E1   -57.870, E3 +255632.465}
SPL {X  -157.825, Y  +713.519, Z    +0.000, E1   -57.630, E3 +255641.701}
SPL {X  -156.079, Y  +719.864, Z    +0.000, E1   -57.324, E3 +255651.664}
SPL {X  -154.064, Y  +726.175, Z    +0.000, E1   -57.042, E3 +255661.426}
SPL {X  -152.053, Y  +731.726, Z    +0.000, E1   -56.648, E3 +255670.711}
SPL {X  -150.108, Y  +736.570, Z    +0.000, E1   -56.283, E3 +255678.950}
SPL {X  -147.726, Y  +741.964, Z    +0.000, E1   -55.884, E3 +255687.986}
SPL {X  -145.163, Y  +747.242, Z    +0.000, E1   -55.517, E3 +255696.582}
SPL {X  -142.489, Y  +752.286, Z    +0.000, E1   -55.227, E3 +255704.409}
SPL {X  -136.074, Y  +762.910, Z    +0.000, E1   -57.336, E3 +255707.531}
SPL {X  -116.561, Y  +787.183, Z    +0.000, E1   -51.088, E3 +255791.999}
ENDSPLINE

SPLINE
SPL {X  -119.623, Y  +783.957, Z    +0.000, E1   -49.202, E3 +255916.532}
SPL {X  -149.958, Y  +736.927, Z    +0.000, E1   -34.772, E3 +255914.249}
SPL {X  -158.826, Y  +709.343, Z    +0.000, E1   -23.029, E3 +255922.592}
SPL {X  -161.800, Y  +691.694, Z    +0.000, E1   -13.520, E3 +255924.886}
SPL {X  -162.597, Y  +682.022, Z    +0.000, E1    -7.544, E3 +255924.542}
SPL {X  -162.813, Y  +675.055, Z    +0.000, E1    -2.911, E3 +255925.184}
SPL {X  -162.820, Y  +671.620, Z    +0.000, E1    -0.225, E3 +255924.696}
SPL {X  -162.820, Y  +669.030, Z    +0.000, E1    +2.242, E3 +255924.397}
SPL {X  -162.820, Y  +664.667, Z    +0.000, E1    +7.867, E3 +255924.100}
SPL {X  -162.820, Y  +660.022, Z    +0.000, E1   +14.535, E3 +255923.997}
SPL {X  -162.820, Y  +653.408, Z    +0.000, E1   +24.221, E3 +255924.307}
SPL {X  -162.820, Y  +640.244, Z    +0.000, E1   +41.042, E3 +255924.351}
SPL {X  -162.820, Y  +592.517, Z    +0.000, E1   +60.575, E3 +255943.482}
SPL {X  -162.820, Y  +515.613, Z    +0.000, E1   +60.751, E3 +256017.317}
ENDSPLINE

SPLINE
SPL {X  -162.820, Y  +518.198, Z    +0.000, E1   +58.338, E3 +256030.473}
ENDSPLINE

SPLINE
SPL {X  -162.820, Y  +508.314, Z    +0.000, E1   +58.337, E3 +256043.169}
SPL {X  -162.820, Y  +498.518, Z    +0.000, E1   +58.346, E3 +256055.675}
SPL {X  -162.820, Y  +489.418, Z    +0.000, E1   +58.357, E3 +256067.265}
SPL {X  -162.820, Y  +479.904, Z    +0.000, E1   +58.389, E3 +256079.312}
SPL {X  -162.820, Y  +472.095, Z    +0.000, E1   +58.202, E3 +256090.492}
SPL {X  -162.820, Y  +463.661, Z    +0.000, E1   +58.370, E3 +256100.278}
SPL {X  -162.820, Y  +454.904, Z    +0.000, E1   +58.380, E3 +256111.444}
SPL {X  -162.820, Y  +446.206, Z    +0.000, E1   +58.278, E3 +256123.335}
SPL {X  -162.820, Y  +436.416, Z    +0.000, E1   +58.325, E3 +256135.575}
SPL {X  -162.820, Y  +426.628, Z    +0.000, E1   +58.432, E3 +256147.443}
SPL {X  -162.820, Y  +418.389, Z    +0.000, E1   +58.300, E3 +256158.846}
SPL {X  -162.820, Y  +412.292, Z    +0.000, E1   +58.070, E3 +256168.214}
SPL {X  -162.820, Y  +403.663, Z    +0.000, E1   +58.258, E3 +256178.154}
SPL {X  -162.820, Y  +397.157, Z    +0.000, E1   +58.054, E3 +256187.890}
SPL {X  -162.820, Y  +387.359, Z    +0.000, E1   +58.365, E3 +256198.519}
SPL {X  -162.810, Y  +378.731, Z    +0.000, E1   +58.366, E3 +256209.577}
SPL {X  -162.546, Y  +371.051, Z    +0.000, E1   +58.239, E3 +256220.297}
SPL {X  -161.863, Y  +362.875, Z    +0.000, E1   +58.273, E3 +256230.522}
SPL {X  -161.159, Y  +357.301, Z    +0.000, E1   +57.946, E3 +256239.822}
SPL {X  -159.864, Y  +349.614, Z    +0.000, E1   +57.922, E3 +256249.898}
SPL {X  -158.300, Y  +342.404, Z    +0.000, E1   +57.579, E3 +256261.344}
SPL {X  -156.187, Y  +334.499, Z    +0.000, E1   +57.331, E3 +256273.004}
SPL {X  -154.237, Y  +328.333, Z    +0.000, E1   +56.930, E3 +256283.214}
SPL {X  -152.732, Y  +324.078, Z    +0.000, E1   +56.482, E3 +256291.219}
SPL {X  -150.609, Y  +318.634, Z    +0.000, E1   +56.366, E3 +256298.913}
SPL {X  -148.206, Y  +313.080, Z    +0.000, E1   +55.888, E3 +256308.625}
SPL {X  -145.956, Y  +308.339, Z    +0.000, E1   +55.380, E3 +256317.301}
SPL {X  -143.330, Y  +303.254, Z    +0.000, E1   +55.057, E3 +256325.421}
SPL {X  -137.431, Y  +293.190, Z    +0.000, E1   +56.809, E3 +256329.584}
SPL {X  -115.845, Y  +266.087, Z    +0.000, E1   +50.276, E3 +256428.442}
SPL {X  -114.083, Y  +264.330, Z    +0.000, E1   +49.123, E3 +256467.152}
ENDSPLINE

SPLINE
SPL {X  -149.622, Y  +316.285, Z    +0.000, E1   +35.036, E3 +256535.664}
SPL {X  -158.704, Y  +344.121, Z    +0.000, E1   +23.312, E3 +256545.537}
SPL {X  -161.701, Y  +361.440, Z    +0.000, E1   +13.961, E3 +256544.608}
SPL {X  -162.691, Y  +374.019, Z    +0.000, E1    +6.263, E3 +256545.261}
SPL {X  -162.820, Y  +380.238, Z    +0.000, E1    +1.925, E3 +256544.945}
SPL {X  -162.820, Y  +383.454, Z    +0.000, E1    -0.619, E3 +256544.551}
SPL {X  -162.820, Y  +387.033, Z    +0.000, E1    -4.758, E3 +256544.255}
SPL {X  -162.820, Y  +390.967, Z    +0.000, E1    -9.918, E3 +256544.700}
SPL {X  -162.820, Y  +397.718, Z    +0.000, E1   -19.761, E3 +256544.074}
SPL {X  -162.820, Y  +405.058, Z    +0.000, E1   -29.962, E3 +256544.987}
SPL {X  -162.820, Y  +417.515, Z    +0.000, E1   -44.878, E3 +256544.149}
SPL {X  -162.820, Y  +462.065, Z    +0.000, E1   -61.507, E3 +256561.109}
SPL {X  -162.820, Y  +504.602, Z    +0.000, E1   -64.286, E3 +256586.635}
SPL {X  -162.820, Y  +535.709, Z    +0.000, E1   -59.182, E3 +256644.314}
SPL {X  -162.820, Y  +543.678, Z    +0.000, E1   -58.515, E3 +256658.703}
SPL {X  -162.820, Y  +553.725, Z    +0.000, E1   -58.454, E3 +256671.964}
SPL {X  -162.820, Y  +562.850, Z    +0.000, E1   -58.373, E3 +256684.126}
SPL {X  -162.820, Y  +573.452, Z    +0.000, E1   -58.444, E3 +256697.339}
SPL {X  -162.820, Y  +583.632, Z    +0.000, E1   -58.444, E3 +256710.266}
SPL {X  -162.820, Y  +591.768, Z    +0.000, E1   -58.375, E3 +256721.130}
SPL {X  -162.820, Y  +601.090, Z    +0.000, E1   -58.519, E3 +256732.117}
SPL {X  -162.820, Y  +609.492, Z    +0.000, E1   -58.431, E3 +256743.422}
SPL {X  -162.820, Y  +617.241, Z    +0.000, E1   -58.340, E3 +256753.947}
SPL {X  -162.820, Y  +626.506, Z    +0.000, E1   -58.420, E3 +256765.329}
SPL {X  -162.820, Y  +635.919, Z    +0.000, E1   -58.604, E3 +256776.073}
SPL {X  -162.820, Y  +643.895, Z    +0.000, E1   -58.380, E3 +256787.838}
SPL {X  -162.820, Y  +653.118, Z    +0.000, E1   -58.401, E3 +256799.435}
SPL {X  -162.820, Y  +660.924, Z    +0.000, E1   -58.393, E3 +256809.503}
SPL {X  -162.820, Y  +670.459, Z    +0.000, E1   -58.489, E3 +256821.104}
SPL {X  -162.713, Y  +679.396, Z    +0.000, E1   -58.414, E3 +256833.003}
SPL {X  -162.301, Y  +686.495, Z    +0.000, E1   -58.302, E3 +256842.787}
SPL {X  -161.571, Y  +693.631, Z    +0.000, E1   -58.186, E3 +256852.751}
SPL {X  -160.411, Y  +701.402, Z    +0.000, E1   -58.100, E3 +256863.227}
SPL {X  -159.229, Y  +707.508, Z    +0.000, E1   -57.870, E3 +256872.465}
SPL {X  -157.825, Y  +713.519, Z    +0.000, E1   -57.630, E3 +256881.701}
SPL {X  -156.079, Y  +719.864, Z    +0.000, E1   -57.324, E3 +256891.664}
SPL {X  -154.064, Y  +726.175, Z    +0.000, E1   -57.042, E3 +256901.426}
SPL {X  -152.053, Y  +731.726, Z    +0.000, E1   -56.648, E3 +256910.711}
SPL {X  -150.108, Y  +736.570, Z    +0.000, E1   -56.283, E3 +256918.950}
SPL {X  -147.726, Y  +741.964, Z    +0.000, E1   -55.884, E3 +256927.986}
SPL {X  -145.163, Y  +747.242, Z    +0.000, E1   -55.517, E3 +256936.582}
SPL {X  -142.489, Y  +752.286, Z    +0.000, E1   -55.227, E3 +256944.409}
SPL {X  -136.074, Y  +762.910, Z    +0.000, E1   -57.336, E3 +256947.531}
SPL {X  -121.244, Y  +782.175, Z    +0.000, E1   -51.023, E3 +257019.476}
SPL {X  -114.422, Y  +789.335, Z    +0.000, E1   -51.094, E3 +257038.092}
ENDSPLINE

SPLINE
SPL {X  -119.623, Y  +783.957, Z    +0.000, E1   -49.202, E3 +257156.532}
SPL {X  -149.958, Y  +736.927, Z    +0.000, E1   -34.772, E3 +257154.249}
SPL {X  -158.826, Y  +709.343, Z    +0.000, E1   -23.029, E3 +257162.592}
SPL {X  -161.800, Y  +691.694, Z    +0.000, E1   -13.520, E3 +257164.886}
SPL {X  -162.711, Y  +679.444, Z    +0.000, E1    -5.922, E3 +257164.960}
SPL {X  -162.820, Y  +673.886, Z    +0.000, E1    -1.998, E3 +257165.121}
SPL {X  -162.820, Y  +670.901, Z    +0.000, E1    +0.338, E3 +257164.555}
SPL {X  -162.820, Y  +667.984, Z    +0.000, E1    +3.594, E3 +257164.387}
SPL {X  -162.820, Y  +664.667, Z    +0.000, E1    +7.867, E3 +257164.100}
SPL {X  -162.820, Y  +660.022, Z    +0.000, E1   +14.535, E3 +257163.997}
SPL {X  -162.820, Y  +653.408, Z    +0.000, E1   +24.221, E3 +257164.307}
SPL {X  -162.820, Y  +640.244, Z    +0.000, E1   +41.042, E3 +257164.351}
SPL {X  -162.820, Y  +602.578, Z    +0.000, E1   +60.061, E3 +257175.766}
SPL {X  -162.820, Y  +586.468, Z    +0.000, E1   +60.779, E3 +257188.168}
SPL {X  -162.820, Y  +515.613, Z    +0.000, E1   +60.751, E3 +257257.317}
ENDSPLINE

SPLINE
SPL {X  -162.820, Y  +518.198, Z    +0.000, E1   +58.338, E3 +257270.473}
ENDSPLINE

